	IF icschange=0 THEN
		AGBControl.eCoordSystem:=L_MC4P_CoordSystem.MCS;//笛卡尔坐标系MCS
		iCurrentCS:=L_MC4P_CoordSystem.MCS;
	END_IF
	IF icschange=1 THEN
		AGBControl.eCoordSystem:=L_MC4P_CoordSystem.ACS;//轴坐标系ACS
		iCurrentCS:=L_MC4P_CoordSystem.MCS;
	END_IF
	IF icschange=2 THEN
		AGBControl.eCoordSystem:=L_MC4P_CoordSystem.PCS_5;//PCS_5
		iCurrentCS:=L_MC4P_CoordSystem.PCS_5;
	END_IF
	IF icschange=4 THEN
		AGBControl.eCoordSystem:=L_MC4P_CoordSystem.PCS_6;//PCS_6
		iCurrentCS:=L_MC4P_CoordSystem.PCS_6;
	END_IF				
	
	AGBControl.axJogPos:=axJogPos;
	AGBControl.axJogNeg:=axJogNeg;
	xBTtest:=BYTE_TO_BOOL(bBTMenu1);
	
	//4. 读取机器人实际位置		
	ReadActPos_ACS.CoordSystem:=L_MC4P_CoordSystem.ACS;
	ReadActPos_ACS.Enable:=TRUE;
	ReadActPos_ACS(AxesGroup:=Delta_Robot);
	
	IF ReadActPos_ACS.Valid=TRUE THEN
		RobotPos.rRobotPosA1:=LREAL_TO_REAL(ReadActPos_ACS.Position[1]);
		RobotPos.rRobotPosA2:=LREAL_TO_REAL(ReadActPos_ACS.Position[2]);
		RobotPos.rRobotPosA3:=LREAL_TO_REAL(ReadActPos_ACS.Position[3]);
	END_IF

	ReadActPos_CS.CoordSystem:=iCurrentCS;
	ReadActPos_CS.Enable:=TRUE;
	ReadActPos_CS(AxesGroup:=Delta_Robot);
	
	IF ReadActPos_CS.Valid=TRUE THEN
		RobotPos.rRobotPosX:=LREAL_TO_REAL(ReadActPos_CS.Position[1]);
		RobotPos.rRobotPosY:=LREAL_TO_REAL(ReadActPos_CS.Position[2]);
		RobotPos.rRobotPosZ:=LREAL_TO_REAL(ReadActPos_CS.Position[3]);
		//RobotPos.rRobotPosC:=LREAL_TO_REAL(ReadActPos_CS.Position[7]);
		//RobotPos.rRobotPosC:=LREAL_TO_REAL(AxisYaw.lrActPosition); //modified in 2016.11.03
	END_IF
		
	//5. 机器人示教
	FOR i:=1 TO iTeachPtNO BY 1 DO				//获取当前位置
		IF bCurrentPos[i]=1 THEN
			aLRPP_TeachPoints[i].X:=RobotPos.rRobotPosX;
			aLRPP_TeachPoints[i].Y:=RobotPos.rRobotPosY;
			aLRPP_TeachPoints[i].Z:=RobotPos.rRobotPosZ;
			aLRPP_TeachPoints[i].C:=RobotPos.rRobotPosC;
			aLRPP_TeachPoints[i].CS_Num:=iCurrentCS;
			bCurrentPos[i]:=0;
		END_IF
	END_FOR
	IF bSavePt=1 THEN
			aLRPP_TeachPoints[iSelectTeNO-4].X:=RobotPos.rRobotPosX;
			aLRPP_TeachPoints[iSelectTeNO-4].Y:=RobotPos.rRobotPosY;
			aLRPP_TeachPoints[iSelectTeNO-4].Z:=RobotPos.rRobotPosZ;
			aLRPP_TeachPoints[iSelectTeNO-4].C:=RobotPos.rRobotPosC;
			aLRPP_TeachPoints[iSelectTeNO-4].CS_Num:=iCurrentCS;
			bSavePt:=0;
	END_IF
	//////////装箱示教////////
	IF xBox_ReadBelt THEN
		rBox_BeltPos:=LREAL_TO_REAL(Outfeeder.lrActPosition);
		xBox_ReadBelt:=FALSE;
	END_IF
	
	IF xBox_Tch THEN
		IF Outfeeder.lrActPosition>rBox_BeltPos THEN
			aLRPP_TeachPoints[iBox_TchNo-4].X:=LREAL_TO_REAL(RobotPos.rRobotPosX-(Outfeeder.lrActPosition-rBox_BeltPos));
		ELSE
			aLRPP_TeachPoints[iBox_TchNo-4].X:=LREAL_TO_REAL(RobotPos.rRobotPosX-(Outfeeder.lrActPosition+Outfeeder.lrcyclelength-rBox_BeltPos));
		END_IF		
		aLRPP_TeachPoints[iBox_TchNo-4].Y:=RobotPos.rRobotPosY;
		aLRPP_TeachPoints[iBox_TchNo-4].Z:=RobotPos.rRobotPosZ;
		aLRPP_TeachPoints[iBox_TchNo-4].C:=RobotPos.rRobotPosC;
		aLRPP_TeachPoints[iBox_TchNo-4].CS_Num:=iCurrentCS;
		xBox_Tch:=0;
	END_IF	

	//装箱体初始化
	p_rBoxLength:=rBoxLength;				//箱体长度
	p_rBoxBiasLength:=rBoxBiasLength;		//箱体偏置长度//产品检测传感器初始化

	p_iNewProdNum:=iNewProdNum;
	//检测产品传感器设置
 
	p_rBoxOutfeederVel:=rBoxOutfeederVel;// 装箱时出料带的速度
	p_rBoxPickTime:=rBoxPickTime;// 装箱抓取物料时间
	p_rBoxPlaceTime:=rBoxPlaceTime;// 装箱放置物料时间
	p_rBoxDetectPosX:=rBoxDetectPosX;// 装箱检测箱体的初始位置     
	p_iBoxTotalPrdoNr:=iBoxTotalPrdoNr;
	//////////装箱示教////////
	
	
	//6. 吸盘标定		

	IF xReadCalibCaxisAngle THEN
		rCalibCaxisAngle:=LREAL_TO_REAL(RobotPos.rRobotPosC);
		rCalibCaxisAngletoRad:=LREAL_TO_REAL(rCalibCaxisAngle*2*Pi/360);
	END_IF

												
	p_iSuckerNum:=iSuckerNum; 	//吸盘标定
	p_iCalibSucker:=iCalibSucker;
	p_rSuker1BiasX:=rSuker1BiasX;
	p_rSuker1BiasY:=rSuker1BiasY;
	p_rSuker2BiasX:=rSuker2BiasX;
	p_rSuker2BiasY:=rSuker2BiasY;
	p_rSuker3BiasX:=rSuker3BiasX;
	p_rSuker3BiasY:=rSuker3BiasY;
	p_rSuker4BiasX:=rSuker4BiasX;
	p_rSuker4BiasY:=rSuker4BiasY;
	//p_rCalibCaxisAngle:=rCalibCaxisAngle;	
		
	IF xToolActive THEN	
		xToolActive:=FALSE;		
	END_IF	
	
	IF 	xToolDeActive THEN
		xToolDeActive:=FALSE;
	END_IF
		
	IF iCalibSucker=0 THEN
		rBiasX:=0;
		rBiasY:=0;	
	END_IF
	IF iCalibSucker=1 THEN
		rBiasX:=rSuker1BiasX;
		rBiasY:=rSuker1BiasY;	
	END_IF
	
	IF iCalibSucker=2 THEN
		rBiasX:=rSuker2BiasX;
		rBiasY:=rSuker2BiasY;	
	END_IF	

	IF iCalibSucker=3 THEN
		rBiasX:=rSuker3BiasX;
		rBiasY:=rSuker3BiasY;				
	END_IF		
	
	IF iCalibSucker=4 THEN
		rBiasX:=rSuker4BiasX;
		rBiasY:=rSuker4BiasY;				
	END_IF	
         
	
	//7. InfeedBeltOrigin坐标系标定
	IF xInfeedRead0=TRUE THEN
		p_rConveyorInRecord0:=rConveyorInRecord0:=LREAL_TO_REAL(Infeeder.lrActPosition);
	END_IF
	p_rConveyorInRecord0:=rConveyorInRecord0;
	
	IF xInfeedRead1=TRUE THEN
		IF Infeeder.lrActPosition<rConveyorInRecord0 THEN
			p_rConveyorInRecord1:=rConveyorInRecord1:=LREAL_TO_REAL(Infeeder.lrActPosition+Infeeder.lrcyclelength);
		ELSE
			p_rConveyorInRecord1:=rConveyorInRecord1:=LREAL_TO_REAL(Infeeder.lrActPosition);
		END_IF		
		p_rReadInfeedPos1_X:=rReadInfeedPos1_X:=LREAL_TO_REAL(RobotPos.rRobotPosX);
		p_rReadInfeedPos1_Y:=rReadInfeedPos1_Y:=LREAL_TO_REAL(RobotPos.rRobotPosY);
		p_rReadInfeedPos1_Z:=rReadInfeedPos1_Z:=LREAL_TO_REAL(RobotPos.rRobotPosZ);
	END_IF
	p_rConveyorInRecord1:=rConveyorInRecord1;
	p_rReadInfeedPos1_X:=rReadInfeedPos1_X;
	p_rReadInfeedPos1_Y:=rReadInfeedPos1_Y;
	p_rReadInfeedPos1_Z:=rReadInfeedPos1_Z;
	
	IF xInfeedRead2=TRUE THEN
		IF Infeeder.lrActPosition<rConveyorInRecord1 THEN
			p_rConveyorInRecord2:=rConveyorInRecord2:=LREAL_TO_REAL(Infeeder.lrActPosition+Infeeder.lrcyclelength);
		ELSE
			p_rConveyorInRecord2:=rConveyorInRecord2:=LREAL_TO_REAL(Infeeder.lrActPosition);
		END_IF

		p_rReadInfeedPos2_X:=rReadInfeedPos2_X:=LREAL_TO_REAL(RobotPos.rRobotPosX);
		p_rReadInfeedPos2_Y:=rReadInfeedPos2_Y:=LREAL_TO_REAL(RobotPos.rRobotPosY);
		p_rReadInfeedPos2_Z:=rReadInfeedPos2_Z:=LREAL_TO_REAL(rReadInfeedPos1_Z);//标定与Z无关，仅取一次Z值		
	END_IF
	
	p_rConveyorInRecord2:=rConveyorInRecord2;
	p_rReadInfeedPos2_X:=rReadInfeedPos2_X;
	p_rReadInfeedPos2_Y:=rReadInfeedPos2_Y;
	p_rReadInfeedPos2_Z:=rReadInfeedPos2_Z;
	
	IF xInfeedRead3=TRUE THEN
		p_rReadInfeedPos3_X:=rReadInfeedPos3_X:=LREAL_TO_REAL(RobotPos.rRobotPosX);
		p_rReadInfeedPos3_Y:=rReadInfeedPos3_Y:=LREAL_TO_REAL(RobotPos.rRobotPosY);
		p_rReadInfeedPos3_Z:=rReadInfeedPos3_Z:=LREAL_TO_REAL(rReadInfeedPos1_Z);//标定与Z无关，仅取一次Z值		
	END_IF
	
	
	p_rReadInfeedPos3_X:=rReadInfeedPos3_X;
	p_rReadInfeedPos3_Y:=rReadInfeedPos3_Y;
	p_rReadInfeedPos3_Z:=rReadInfeedPos3_Z;
	
	IF xInfeedRead4=TRUE THEN
		p_rReadInfeedPos4_X:=rReadInfeedPos4_X:=LREAL_TO_REAL(RobotPos.rRobotPosX);
		p_rReadInfeedPos4_Y:=rReadInfeedPos4_Y:=LREAL_TO_REAL(RobotPos.rRobotPosY);
		p_rReadInfeedPos4_Z:=rReadInfeedPos4_Z:=LREAL_TO_REAL(rReadInfeedPos1_Z);//标定与Z无关，仅取一次Z值		
	END_IF
	
	p_rReadInfeedPos4_X:=rReadInfeedPos4_X;
	p_rReadInfeedPos4_Y:=rReadInfeedPos4_Y;
	p_rReadInfeedPos4_Z:=rReadInfeedPos4_Z;		

	//计算传动带（进料带）原点并标定PCS5（InS）
	IF xCaculateInfeedBeltOrigin=TRUE THEN
		
		FourPts_Calibration_1(
			rReadfeedPos1_X:= rReadInfeedPos1_X, 
			rReadfeedPos1_Y:= rReadInfeedPos1_Y, 
			rReadfeedPos1_Z:= rReadInfeedPos1_Z, 
			rReadfeedPos2_X:= rReadInfeedPos2_X, 
			rReadfeedPos2_Y:= rReadInfeedPos2_Y, 
			rReadfeedPos3_X:= rReadInfeedPos3_X, 
			rReadfeedPos3_Y:= rReadInfeedPos3_Y, 
			rReadfeedPos4_X:= rReadInfeedPos4_X, 
			rReadfeedPos4_Y:= rReadInfeedPos4_Y, 
			rRotation_C=> sInFeedBeltOrigin.rRotation_C,
			Output_X0=>PCS5_X0	,
			Output_Y0=>PCS5_Y0	,	
			Output_X1=>PCS5_X1	,	
			Output_Y1=>PCS5_Y1	,	
			Output_X2=>PCS5_X2	,	
			Output_Y2=>PCS5_Y2	,	
			Output_X3=>PCS5_X3	,	
			Output_Y3=>PCS5_Y3	,	
			dx=>PCS5_dx	,			
			dy=>PCS5_dy	,	);
			  	
		p_PCS5_X0:=PCS5_X0;
		p_PCS5_Y0:=PCS5_Y0;
		p_PCS5_X1:=PCS5_X1;
		p_PCS5_Y1:=PCS5_Y1;
		p_PCS5_X2:=PCS5_X2;
		p_PCS5_Y2:=PCS5_Y2;
		p_PCS5_X3:=PCS5_X3;
		p_PCS5_Y3:=PCS5_Y3;
		p_PCS5_dx:=PCS5_dx;
		p_PCS5_dy:=PCS5_dy;
		
		//p_sInFeedBeltOrigin.rOriginPosX:=sInFeedBeltOrigin.rOriginPosX:=rReadInfeedPos1_X;
		//p_sInFeedBeltOrigin.rOriginPosY:=sInFeedBeltOrigin.rOriginPosY:=rReadInfeedPos1_Y;
		p_sInFeedBeltOrigin.rOriginPosX:=sInFeedBeltOrigin.rOriginPosX:=(rReadInfeedPos1_X+rReadInfeedPos2_X+rReadInfeedPos3_X+rReadInfeedPos4_X)/4.0;
		p_sInFeedBeltOrigin.rOriginPosY:=sInFeedBeltOrigin.rOriginPosY:=(rReadInfeedPos1_Y+rReadInfeedPos2_Y+rReadInfeedPos3_Y+rReadInfeedPos4_Y)/4.0;
		
		p_sInFeedBeltOrigin.rOriginPosZ:=sInFeedBeltOrigin.rOriginPosZ:=rReadInfeedPos1_Z;
		p_sInFeedBeltOrigin.rRotation_C:=sInFeedBeltOrigin.rRotation_C;
						
		//开始标定InS（PCS5）			
		fbPCS5_Calib.TransX:=p_PCS5_OriginX:=PCS5_OriginX:=	p_sInFeedBeltOrigin.rOriginPosX;
		fbPCS5_Calib.TransY:=p_PCS5_OriginY:=PCS5_OriginY:=	p_sInFeedBeltOrigin.rOriginPosY;
		fbPCS5_Calib.TransZ:=p_PCS5_OriginZ:=PCS5_OriginZ:=	p_sInFeedBeltOrigin.rOriginPosZ;
		fbPCS5_Calib.RotAngle1:=p_PCS5_OriginA:=PCS5_OriginA:=	p_sInFeedBeltOrigin.rRotation_A;
		fbPCS5_Calib.RotAngle2:=p_PCS5_OriginB:=PCS5_OriginB:=	p_sInFeedBeltOrigin.rRotation_B;
		fbPCS5_Calib.RotAngle3:=p_PCS5_OriginC:=PCS5_OriginC:=	p_sInFeedBeltOrigin.rRotation_C;
		fbPCS5_Calib.Execute:=TRUE;
		fbPCS5_Calib.CoordSystem:=L_MC4P_CoordSystem.PCS_5;	
		xCaculateInfeedBeltOrigin:=FALSE;
		
	END_IF
	
	IF fbPCS5_Calib.Done=TRUE THEN
		fbPCS5_Calib.Execute:=FALSE;
	END_IF			
	fbPCS5_Calib(AxesGroup:=Delta_Robot);

	
	//再次将标定值赋给Pst，以便用户自修改	
	p_sInFeedBeltOrigin.rOriginPosX:=sInFeedBeltOrigin.rOriginPosX; //传动带原点
	p_sInFeedBeltOrigin.rOriginPosY:=sInFeedBeltOrigin.rOriginPosY;
	p_sInFeedBeltOrigin.rOriginPosZ:=sInFeedBeltOrigin.rOriginPosZ;
	p_sInFeedBeltOrigin.rRotation_A:=sInFeedBeltOrigin.rRotation_A;
	p_sInFeedBeltOrigin.rRotation_B:=sInFeedBeltOrigin.rRotation_B;
	p_sInFeedBeltOrigin.rRotation_C:=sInFeedBeltOrigin.rRotation_C;
	
			
	//8. OutfeedBeltOrigin坐标系标定 Outfeeder是出料带
	IF xOutfeedRead0=TRUE THEN
		p_rConveyorOutRecord0:=rConveyorOutRecord0:=LREAL_TO_REAL(Outfeeder.lrActPosition);
	END_IF
	
	p_rConveyorOutRecord0:=rConveyorOutRecord0;
	
	IF xOutfeedRead1=TRUE THEN
		IF Outfeeder.lrActPosition<rConveyorOutRecord0 THEN
			p_rConveyorOutRecord1:=rConveyorOutRecord1:=LREAL_TO_REAL(Outfeeder.lrActPosition+Outfeeder.lrcyclelength);
		ELSE
			p_rConveyorOutRecord1:=rConveyorOutRecord1:=LREAL_TO_REAL(Outfeeder.lrActPosition);
		END_IF	
		p_rReadOutfeedPos1_X:=rReadOutfeedPos1_X:=LREAL_TO_REAL(RobotPos.rRobotPosX);
		p_rReadOutfeedPos1_Y:=rReadOutfeedPos1_Y:=LREAL_TO_REAL(RobotPos.rRobotPosY);
		p_rReadOutfeedPos1_Z:=rReadOutfeedPos1_Z:=LREAL_TO_REAL(RobotPos.rRobotPosZ);
	END_IF
	p_rConveyorOutRecord1:=rConveyorOutRecord1;
	p_rReadOutfeedPos1_X:=rReadOutfeedPos1_X;
	p_rReadOutfeedPos1_Y:=rReadOutfeedPos1_Y;
	p_rReadOutfeedPos1_Z:=rReadOutfeedPos1_Z;		
	                            
	IF xOutfeedRead2=TRUE THEN
		IF Outfeeder.lrActPosition<rConveyorOutRecord1 THEN
			p_rConveyorOutRecord2:=rConveyorOutRecord2:=LREAL_TO_REAL(Outfeeder.lrActPosition+Outfeeder.lrcyclelength);
		ELSE
			p_rConveyorOutRecord2:=rConveyorOutRecord2:=LREAL_TO_REAL(Outfeeder.lrActPosition);
		END_IF	

		p_rReadOutfeedPos2_X:=rReadOutfeedPos2_X:=LREAL_TO_REAL(RobotPos.rRobotPosX);
		p_rReadOutfeedPos2_Y:=rReadOutfeedPos2_Y:=LREAL_TO_REAL(RobotPos.rRobotPosY);
		p_rReadOutfeedPos2_Z:=rReadOutfeedPos2_Z:=LREAL_TO_REAL(rReadOutfeedPos1_Z);//标定与Z无关，仅取一次Z值
	END_IF
	p_rConveyorOutRecord2:=rConveyorOutRecord2;
	p_rReadOutfeedPos2_X:=rReadOutfeedPos2_X;
	p_rReadOutfeedPos2_Y:=rReadOutfeedPos2_Y;	
	p_rReadOutfeedPos2_Z:=rReadOutfeedPos2_Z;	
	
	IF xOutfeedRead3=TRUE THEN
		p_rReadOutfeedPos3_X:=rReadOutfeedPos3_X:=LREAL_TO_REAL(RobotPos.rRobotPosX);
		p_rReadOutfeedPos3_Y:=rReadOutfeedPos3_Y:=LREAL_TO_REAL(RobotPos.rRobotPosY);
		p_rReadOutfeedPos3_Z:=rReadOutfeedPos3_Z:=LREAL_TO_REAL(rReadOutfeedPos1_Z);//标定与Z无关，仅取一次Z值
	END_IF

	p_rReadOutfeedPos3_X:=rReadOutfeedPos3_X;
	p_rReadOutfeedPos3_Y:=rReadOutfeedPos3_Y;	
	p_rReadOutfeedPos3_Z:=rReadOutfeedPos3_Z;	
	
	IF xOutfeedRead4=TRUE THEN
		p_rReadOutfeedPos4_X:=rReadOutfeedPos4_X:=LREAL_TO_REAL(RobotPos.rRobotPosX);
		p_rReadOutfeedPos4_Y:=rReadOutfeedPos4_Y:=LREAL_TO_REAL(RobotPos.rRobotPosY);
		p_rReadOutfeedPos4_Z:=rReadOutfeedPos4_Z:=LREAL_TO_REAL(rReadOutfeedPos1_Z);//标定与Z无关，仅取一次Z值
	END_IF
	
	p_rReadOutfeedPos4_X:=rReadOutfeedPos4_X;
	p_rReadOutfeedPos4_Y:=rReadOutfeedPos4_Y;	
	p_rReadOutfeedPos4_Z:=rReadOutfeedPos4_Z;	

	
	//计算传动带（出料带）原点并标定PCS6（OtS）
	IF	xCaculateOutfeedBeltOrigin=TRUE THEN
		
			FourPts_Calibration_2(
					rReadfeedPos1_X:= rReadOutfeedPos1_X, 
					rReadfeedPos1_Y:= rReadOutfeedPos1_Y, 
					rReadfeedPos1_Z:= rReadOutfeedPos1_Z, 
					rReadfeedPos2_X:= rReadOutfeedPos2_X, 
					rReadfeedPos2_Y:= rReadOutfeedPos2_Y, 
					rReadfeedPos3_X:= rReadOutfeedPos3_X, 
					rReadfeedPos3_Y:= rReadOutfeedPos3_Y, 
					rReadfeedPos4_X:= rReadOutfeedPos4_X, 
					rReadfeedPos4_Y:= rReadOutfeedPos4_Y, 
					rRotation_C=> sOutFeedBeltOrigin.rRotation_C,
					Output_X0=>PCS6_X0	,
                    Output_Y0=>PCS6_Y0	,	
                    Output_X1=>PCS6_X1	,	
                    Output_Y1=>PCS6_Y1	,	
                    Output_X2=>PCS6_X2	,	
                    Output_Y2=>PCS6_Y2	,	
                    Output_X3=>PCS6_X3	,	
                    Output_Y3=>PCS6_Y3	,	
               		dx=>PCS6_dx	,			
			        dy=>PCS6_dy	,	);
			  	
			p_PCS6_X0:=PCS6_X0;
			p_PCS6_Y0:=PCS6_Y0;
			p_PCS6_X1:=PCS6_X1;
			p_PCS6_Y1:=PCS6_Y1;
			p_PCS6_X2:=PCS6_X2;
			p_PCS6_Y2:=PCS6_Y2;
			p_PCS6_X3:=PCS6_X3;
			p_PCS6_Y3:=PCS6_Y3;
			p_PCS6_dx:=PCS6_dx;
			p_PCS6_dy:=PCS6_dy;
			
			p_sOutFeedBeltOrigin.rOriginPosX:=sOutFeedBeltOrigin.rOriginPosX:=(rReadOutfeedPos1_X+rReadOutfeedPos2_X+rReadOutfeedPos3_X+rReadOutfeedPos4_X)/4.0;
			p_sOutFeedBeltOrigin.rOriginPosY:=sOutFeedBeltOrigin.rOriginPosY:=(rReadOutfeedPos1_Y+rReadOutfeedPos2_Y+rReadOutfeedPos3_Y+rReadOutfeedPos4_Y)/4.0;
			//p_sOutFeedBeltOrigin.rOriginPosX:=sOutFeedBeltOrigin.rOriginPosX:=rReadOutfeedPos1_X;
			//p_sOutFeedBeltOrigin.rOriginPosY:=sOutFeedBeltOrigin.rOriginPosY:=rReadOutfeedPos1_Y;
			p_sOutFeedBeltOrigin.rOriginPosZ:=sOutFeedBeltOrigin.rOriginPosZ:=rReadOutfeedPos1_Z;
			p_sOutFeedBeltOrigin.rRotation_C:=sOutFeedBeltOrigin.rRotation_C;
			
			//开始标定InS（PCS5）
			fbPCS6_Calib.TransX:=p_PCS6_OriginX:=PCS6_OriginX:=p_sOutFeedBeltOrigin.rOriginPosX;
			fbPCS6_Calib.TransY:=p_PCS6_OriginY:=PCS6_OriginY:=p_sOutFeedBeltOrigin.rOriginPosY;
			fbPCS6_Calib.TransZ:=p_PCS6_OriginZ:=PCS6_OriginZ:=p_sOutFeedBeltOrigin.rOriginPosZ;
			fbPCS6_Calib.RotAngle1:=p_PCS6_OriginA:=PCS6_OriginA:=p_sOutFeedBeltOrigin.rRotation_A;
			fbPCS6_Calib.RotAngle2:=p_PCS6_OriginB:=PCS6_OriginB:=p_sOutFeedBeltOrigin.rRotation_B;
			fbPCS6_Calib.RotAngle3:=p_PCS6_OriginC:=PCS6_OriginC:=p_sOutFeedBeltOrigin.rRotation_C;
			fbPCS6_Calib.Execute:=TRUE;
			fbPCS6_Calib.CoordSystem:=L_MC4P_CoordSystem.PCS_6;	
			xCaculateOutfeedBeltOrigin:=FALSE;
			
	END_IF
	
	IF fbPCS6_Calib.Done=TRUE THEN
		fbPCS6_Calib.Execute:=FALSE;
	END_IF
	fbPCS6_Calib(AxesGroup:=Delta_Robot);	
	//出料带标定模块
	
	
	
	//再次将标定值赋给Pst，以便用户自修改	
	p_sOutFeedBeltOrigin.rOriginPosX:=sOutFeedBeltOrigin.rOriginPosX; //传动带原点
	p_sOutFeedBeltOrigin.rOriginPosY:=sOutFeedBeltOrigin.rOriginPosY;
	p_sOutFeedBeltOrigin.rOriginPosZ:=sOutFeedBeltOrigin.rOriginPosZ;
	p_sOutFeedBeltOrigin.rRotation_A:=sOutFeedBeltOrigin.rRotation_A;
	p_sOutFeedBeltOrigin.rRotation_B:=sOutFeedBeltOrigin.rRotation_B;
	p_sOutFeedBeltOrigin.rRotation_C:=sOutFeedBeltOrigin.rRotation_C;

	//9. 相机标定界面
	IF xTeachRCalPt2 THEN
		p_RobotCalPt2.rX:=RobotCalPt2.rX:=RobotPos.rRobotPosX+rInfeedMapX;
		p_RobotCalPt2.rY:=RobotCalPt2.rY:=RobotPos.rRobotPosY+rInfeedMapY;
		p_RobotCalPt2.rZ:=RobotCalPt2.rZ:=RobotPos.rRobotPosZ;		
	END_IF
	
	IF xTeachRCalPt3 THEN
		p_RobotCalPt3.rX:=RobotCalPt3.rX:=RobotPos.rRobotPosX+rInfeedMapX;
		p_RobotCalPt3.rY:=RobotCalPt3.rY:=RobotPos.rRobotPosY+rInfeedMapY;
		p_RobotCalPt3.rZ:=RobotCalPt3.rZ:=RobotPos.rRobotPosZ;		
	END_IF																	
	IF xTeachRCalPt4 THEN
		p_RobotCalPt4.rX:=RobotCalPt4.rX:=RobotPos.rRobotPosX+rInfeedMapX;
		p_RobotCalPt4.rY:=RobotCalPt4.rY:=RobotPos.rRobotPosY+rInfeedMapY;
		p_RobotCalPt4.rZ:=RobotCalPt4.rZ:=RobotPos.rRobotPosZ;		
	END_IF	
	
	IF xCaculateCameraCalPts THEN
		
		p_CameraCalPt1.rX:=CameraCalPt1.rX:=(RobotCalPt1.rX-sInFeedBeltOrigin.rOriginPosX)*COS(alpha)+(RobotCalPt1.rY-sInFeedBeltOrigin.rOriginPosY)*SIN(alpha)-(rConveyorInRecord2-rConveyorInRecord0);
		p_CameraCalPt1.rY:=CameraCalPt1.rY:=(-RobotCalPt1.rX+sInFeedBeltOrigin.rOriginPosX)*SIN(alpha)+(RobotCalPt1.rY-sInFeedBeltOrigin.rOriginPosY)*COS(alpha);//-(rConveyorInRecord2-rConveyorInRecord0);
		p_CameraCalPt1.rZ:=CameraCalPt1.rZ:=0;
		
		p_CameraCalPt2.rX:=CameraCalPt2.rX:=(RobotCalPt2.rX-sInFeedBeltOrigin.rOriginPosX)*COS(alpha)+(RobotCalPt2.rY-sInFeedBeltOrigin.rOriginPosY)*SIN(alpha)-(rConveyorInRecord2-rConveyorInRecord0);
		p_CameraCalPt2.rY:=CameraCalPt2.rY:=(-RobotCalPt2.rX+sInFeedBeltOrigin.rOriginPosX)*SIN(alpha)+(RobotCalPt2.rY-sInFeedBeltOrigin.rOriginPosY)*COS(alpha);//-(rConveyorInRecord2-rConveyorInRecord0);
		p_CameraCalPt2.rZ:=CameraCalPt2.rZ:=0;
		
		p_CameraCalPt3.rX:=CameraCalPt3.rX:=(RobotCalPt3.rX-sInFeedBeltOrigin.rOriginPosX)*COS(alpha)+(RobotCalPt3.rY-sInFeedBeltOrigin.rOriginPosY)*SIN(alpha)-(rConveyorInRecord2-rConveyorInRecord0);
		p_CameraCalPt3.rY:=CameraCalPt3.rY:=(-RobotCalPt3.rX+sInFeedBeltOrigin.rOriginPosX)*SIN(alpha)+(RobotCalPt3.rY-sInFeedBeltOrigin.rOriginPosY)*COS(alpha);//-(rConveyorInRecord2-rConveyorInRecord0);
		p_CameraCalPt3.rZ:=CameraCalPt3.rZ:=0;
		
		p_CameraCalPt4.rX:=CameraCalPt4.rX:=(RobotCalPt4.rX-sInFeedBeltOrigin.rOriginPosX)*COS(alpha)+(RobotCalPt4.rY-sInFeedBeltOrigin.rOriginPosY)*SIN(alpha)-(rConveyorInRecord2-rConveyorInRecord0);
		p_CameraCalPt4.rY:=CameraCalPt4.rY:=(-RobotCalPt4.rX+sInFeedBeltOrigin.rOriginPosX)*SIN(alpha)+(RobotCalPt4.rY-sInFeedBeltOrigin.rOriginPosY)*COS(alpha);//-(rConveyorInRecord2-rConveyorInRecord0);
		p_CameraCalPt4.rZ:=CameraCalPt4.rZ:=0;
	
	END_IF
		
END_IF		

(*

IF xAutoRun  or xJumpOutManualJog THEN
	wstep:=5;//返回待机状态
	xJumpOutManualJog:=FALSE;
END_IF

*)
END_ACTION

ACTION A30_AutoRun:
	CustomerPrgHandling.xEnable:=xAutoRun;
IF xAutoRun THEN
	IF iSelfadaptPickSwitch=1 THEN
		lrMaxTimeforCycleAdaptive:=1.0;
	ELSE
		lrMaxTimeforCycleAdaptive:=0.0;
	END_IF
	// 抓取节拍自适应计算
	
	//传送带滤波处理
	L_USPP_PT1Filter_0(
		lrIn:= , 
		lrDelayTime:=1.0 , 
		lrOut=> lrInfeederFilterVelocity, 
		xError=> , 
		eErrorID=> );		
	lrDistToMinCapLForCycleAdaptive:=lrInfeederFilterVelocity*lrMaxTimeforCycleAdaptive;		
	//传送带滤波处理
	
	p_xExternalMode:=xExternalMode;//将外部数据发送模式赋值到断电保持变量 3.1
	
	p_xLocal_or_Remote:=xLocal_or_Remote; //机器人本机控制 or 远程控制
	
	IF fb_PlaceCounter_Triger.Q THEN
		iPlaceCounter:=iPlaceCounter+1;
	END_IF
	
	//托盘的x、y方向间距设置===================2017.12.13============================
		CustomerPrgHandling.rPalletPickDeltaX:=PCS5_dx;
		CustomerPrgHandling.rPalletPickDeltaY:=PCS5_dy;
		CustomerPrgHandling.rPalletPlaceDeltaX:=PCS6_dx;
		CustomerPrgHandling.rPalletPlaceDeltaY:=PCS6_dy;
	//托盘的x、y方向间距设置===================2017.12.13============================	
		
	//抓取线和放置线的计算
	rMinCaptureLine:=CustomerPrg.Table_Position[5].X;
	rMaxCaptureLine:=CustomerPrg.Table_Position[6].X;
	rMinPlaceLine:=CustomerPrg.Table_Position[7].X;
	rMaxPlaceLine:=CustomerPrg.Table_Position[8].X;
	//产品信息
	rProductAdd_Z:=CustomerPrg.Table_Position[9].Z;			
	rFilterTolerance_X:=CustomerPrg.Table_Position[9].X;
	rFilterTolerance_Y:=CustomerPrg.Table_Position[9].Y;	
	
	
	//程序解析运动函数
	//程序解析模块输入	
	//2017.03.30  PnP Cycle Adaptive Fuction
	CustomerPrgHandling.lrDistToMinCapLForCycleAdaptive:=lrDistToMinCapLForCycleAdaptive;
	CustomerPrgHandling.lrMinCaptureLine:= rMinCaptureLine;
	CustomerPrgHandling.lrMaxCaptureLine:= rMaxCaptureLine; 
	
	(*
	CustomerPrgHandling.rCoefMaxOfStartAndEndR[1]:=CoefMaxOfStartAndEndR[1];
	CustomerPrgHandling.iAux1ExePointPassed[1]:=Aux1ExePointPassed[1];		
	CustomerPrgHandling.rAux1DurationRatio[1]:=Aux1DurationRatio[1];				
	CustomerPrgHandling.iAux1MotionLaw[1]:=Aux1MotionLaw[1];				
	CustomerPrgHandling.rStartAlphaRatio[1,1]:=StartAlphaRatio[1,1];	
	CustomerPrgHandling.rStartAlphaRatio[1,2]:=StartAlphaRatio[1,2];
	CustomerPrgHandling.rStartAlphaRatio[1,3]:=StartAlphaRatio[1,3];		
	CustomerPrgHandling.rEndAlphaRatio[1,7]:=EndAlphaRatio[1,7];
	CustomerPrgHandling.rEndAlphaRatio[1,8]:=EndAlphaRatio[1,8];
	CustomerPrgHandling.rEndAlphaRatio[1,9]:=EndAlphaRatio[1,9];
	
	CustomerPrgHandling.rCoefMaxOfStartAndEndR[2]:= CoefMaxOfStartAndEndR[2];
	CustomerPrgHandling.iAux1ExePointPassed[2]:= Aux1ExePointPassed[2];		
	CustomerPrgHandling.rAux1DurationRatio[2]:= Aux1DurationRatio[2];				
	CustomerPrgHandling.iAux1MotionLaw[2]:=Aux1MotionLaw[2];				
	CustomerPrgHandling.rStartAlphaRatio[2,1]:=StartAlphaRatio[2,1];	
	CustomerPrgHandling.rStartAlphaRatio[2,2]:=StartAlphaRatio[2,2];
	CustomerPrgHandling.rStartAlphaRatio[2,3]:=StartAlphaRatio[2,3];		
	CustomerPrgHandling.rEndAlphaRatio[2,7]:=EndAlphaRatio[2,7];
	CustomerPrgHandling.rEndAlphaRatio[2,8]:=EndAlphaRatio[2,8];
	CustomerPrgHandling.rEndAlphaRatio[2,9]:=EndAlphaRatio[2,9];
	*)
		
	CustomerPrgHandling.xDetectBoxSwitch:=DI_3;
	CustomerPrgHandling.CustomerPrg:=CustomerPrg;
	CustomerPrgHandling.xRunInter:=xRunInter;
	CustomerPrgHandling.xStopInter:=xStopInter;
	CustomerPrgHandling.sInFeedBeltOrigin:=	sInFeedBeltOrigin;	
	CustomerPrgHandling.sOutFeedBeltOrigin:=sOutFeedBeltOrigin;                                                            
	//CustomerPrgHandling.lrCurrentAuxC:=AxisYaw.lrActPosition;
	CustomerPrgHandling.rFollowBias_X:=rFollowBias_X;//1
	CustomerPrgHandling.rFollowBias_Y:=rFollowBias_Y;//2
	CustomerPrgHandling.rSuckerDropHeight:=rSuckerDropHeight;//3
	CustomerPrgHandling.rInfeedClutchPra:=rBelt1_ClutchPra;//4
	CustomerPrgHandling.rOutfeedClutchPra:=rBelt2_ClutchPra;//5
	CustomerPrgHandling.rBlowOpenTime:=	rBlow_Gas_OpenTime;//6
	CustomerPrgHandling.rSuckOpenTime:=rSuck_Gas_OpenTime;//7
	CustomerPrgHandling.rBlowGasTime:=rBlowGasTime;//8	
	CustomerPrgHandling.iBox_ExceptionDeal:=iBox_ExceptionDeal;//9
	CustomerPrgHandling.iSelfadaptPickSwitch:=iSelfadaptPickSwitch;//10
	CustomerPrgHandling.rPnPDurationNegativeLimit:=rPnPDurationNegativeLimit;
	CustomerPrgHandling.rPnPDurationPositiveLimit:=rPnPDurationPositiveLimit;	
	CustomerPrgHandling.iProdDeformation:=iProdDeformation; //11 产品变形量	

	CustomerPrgHandling.rProductAdd_Z:=rProductAdd_Z;
	CustomerPrgHandling.rBoxLength:=rBoxLength;
	CustomerPrgHandling.rBoxBiasLength:=rBoxBiasLength;
	
	CustomerPrgHandling.iNewProdNum:=iNewProdNum;//检测物体需要的外部触发信号数量
	
	IF iPrdtDetectDevice=Detect_Device.Camera THEN//产品检测装置选择 	0：相机；1：传感器；2：上位机通讯指定	 可以定义成枚举类型
		IF iSuckerNum <=5 THEN
			CustomerPrgHandling.xProdInfoReady:=BufferHandling.xProdInfoReady;
			CustomerPrgHandling.lrInfeedDeltaX:=BufferHandling.sFirstProdInfo.lrDeltaX;
			CustomerPrgHandling.lrInfeedDeltaY:=BufferHandling.sFirstProdInfo.lrDeltaY;
			CustomerPrgHandling.lrPosAuxC:=BufferHandling.sFirstProdInfo.lrPosAuxC;			
		ELSIF iSuckerNum >=6 THEN		
			CustomerPrgHandling.xProdInfoReady:=MultiPickHandling.xProdGroupReady AND MultiPickHandling.xProdInfoReady;			
			CustomerPrgHandling.lrInfeedDeltaX:=MultiPickHandling.sProductInfo.lrDeltaX;
			CustomerPrgHandling.lrInfeedDeltaY:=MultiPickHandling.sProductInfo.lrDeltaY;
			CustomerPrgHandling.lrPosAuxC:=MultiPickHandling.sProductInfo.lrPosAuxC;		
		END_IF	
	END_IF
	
	IF iPrdtDetectDevice=Detect_Device.Sensor THEN//产品检测装置选择 0：相机；1：传感器；2：上位机通讯指定	
		CustomerPrgHandling.xProdInfoReady:=SensorBufferHandler.xProdInfoReady;
		CustomerPrgHandling.lrInfeedDeltaX:=SensorBufferHandler.sFirstProdInfo.lrDeltaX;
		CustomerPrgHandling.lrInfeedDeltaY:=SensorBufferHandler.sFirstProdInfo.lrDeltaY;
		CustomerPrgHandling.lrPosAuxC:=SensorBufferHandler.sFirstProdInfo.lrPosAuxC;
	END_IF
	
	//程序解析模块输出
	iCommandType							:=CustomerPrgHandling.iCommandType;
	iCurrentPrgCmdNum						:=CustomerPrgHandling.iCurrentPrgCmdNum;
	LoadDistribution.lrFilterTolerance		:=rFilterTolerance_X; //滤波参数
	
	BufferHandling.xFirstProdDel			:=CustomerPrgHandling.xFirstProdDel;
	BufferHandling.lrPaPDuration			:=CustomerPrgHandling.lrPaPDuration;	
	BufferHandling.lrMinCaptureLine			:=rMinCaptureLine;	//抓取起始线	
	BufferHandling.lrMaxCaptureLine			:=rMaxCaptureLine;	//抓取起始线     	
	
	MultiPickHandling.xProductDel			:=CustomerPrgHandling.xFirstProdDel;
	MultiPickHandling.lrPaPDuration			:=CustomerPrgHandling.lrPaPDuration;
	MultiPickHandling.lrMinCaptureLine		:=rMinCaptureLine;	//抓取线限位1 
	MultiPickHandling.lrMaxCaptureLine		:=rMaxCaptureLine;	//抓取线限位2
	MultiPickHandling.lrToleranceDistance	:=500;
	MultiPickHandling.iNrOfTool				:=iSuckerNum;
	
	(*
	xProdInfoReady_TON(IN:=MultiPickHandling.xProdInfoReady,Pt:=T#50MS);
	IF xProdInfoReady_TON.Q THEN
		MultiPickHandling.xProductDel:=TRUE;	
	END_IF
	xProductDel_TON(IN:=MultiPickHandling.xProductDel,Pt:=T#4MS);
	IF xProductDel_TON.Q THEN
		MultiPickHandling.xProductDel:=FALSE;
	END_IF
	*)
	
	//吸气/吹气
	//x_Suck1:=CustomerPrgHandling.xSuck;
	//x_Blow1:=CustomerPrgHandling.xBlow;
	IF xAutoRun THEN
		x_Suck1_HMI:=FALSE;
		x_Blow1_HMI:=FALSE;
	END_IF
	
	
	//传感器检测输入
	SensorBufferHandler.lrMinPickLine:=rMinCaptureLine;
	SensorBufferHandler.lrMaxPickLine:=rMaxCaptureLine;
	SensorBufferHandler.lrPaPDuration:=CustomerPrgHandling.lrPaPDuration;
	SensorBufferHandler.xFirstProdDel:=CustomerPrgHandling.xFirstProdDel;
	
	//传入工具坐标系参数
	CustomerPrgHandling.Tool[1].X:=rSuker1BiasX;
	CustomerPrgHandling.Tool[1].Y:=rSuker1BiasY;
	CustomerPrgHandling.Tool[1].C:=rSuker1PickC;
	//CustomerPrgHandling.Tool[1].Z:=iSuckerHeight;
	CustomerPrgHandling.Tool[2].X:=rSuker2BiasX;
	CustomerPrgHandling.Tool[2].Y:=rSuker2BiasY;
	CustomerPrgHandling.Tool[2].C:=rSuker2PickC;
	//CustomerPrgHandling.Tool[2].Z:=iSuckerHeight;
	CustomerPrgHandling.Tool[3].X:=rSuker3BiasX;
	CustomerPrgHandling.Tool[3].Y:=rSuker3BiasY;
	CustomerPrgHandling.Tool[3].C:=rSuker3PickC;
	//CustomerPrgHandling.Tool[3].Z:=iSuckerHeight;
	CustomerPrgHandling.Tool[4].X:=rSuker4BiasX;
	CustomerPrgHandling.Tool[4].Y:=rSuker4BiasY;
	CustomerPrgHandling.Tool[4].C:=rSuker4PickC;
	//CustomerPrgHandling.Tool[4].Z:=iSuckerHeight;
	
	//保存自动运行参数
	IF xSaveRunPra THEN
		CustomerPrgEdit.SaveRunPra(axSavePrgNo:=p_axSavePrgNo,adr_iCurrentPrgNum:=p_iCurrentPrgNum,xSaveRunPra:=xSaveRunPra,
			rFollowBias_X:=rFollowBias_X,rFollowBias_Y:=rFollowBias_Y,rSuckerDropHeight:=rSuckerDropHeight,
			rBelt1_ClutchPra:=rBelt1_ClutchPra,rBelt2_ClutchPra:=rBelt2_ClutchPra,
			rSuck_Gas_OpenTime:=rSuck_Gas_OpenTime,rBlow_Gas_OpenTime:=rBlow_Gas_OpenTime,rBlowGasTime:=rBlowGasTime,
			iBox_ExceptionDeal:=iBox_ExceptionDeal,
			iSelfadaptPickSwitch:=iSelfadaptPickSwitch,
			rPnPDurationNegativeLimit:=rPnPDurationNegative,
			rPnPDurationPositiveLimit:=rPnPDurationPositive,
			iProdDeformation:=iProdDeformation,
			CustomerPrg:=CustomerPrg,aLRPP_TeachPoints:=aLRPP_TeachPoints);
			
			p_rPnPDurationNegativeLimit:=rPnPDurationNegativeLimit;			
			p_rPnPDurationPositiveLimit:=rPnPDurationPositiveLimit;	
			p_rTorqueForwardControl:=rTorqueForwardControl;	
	END_IF
		
END_IF


//自动运行隐藏主菜单延迟设置	
IF xRunOrStopPrg THEN
	xAutoMenu:=TRUE;
END_IF
DetectStop_Ftrig(CLK:=xRunOrStopPrg, Q=>);
	
IF DetectStop_Ftrig.Q THEN
	fb_TON_Menu.IN:=TRUE;
	fb_TON_Menu.PT:= T#2S; 
END_IF
	
IF fb_TON_Menu.Q=TRUE THEN
	fb_TON_Menu.IN:=FALSE;
	xAutoMenu:=FALSE;
END_IF		
fb_TON_Menu();

//自动运行隐藏主菜单延迟设置	
IF NOT xAutoRun THEN
	iCurrentPrgCmdNum:=1;
	iCommandType:=0;
	iAutoStep:=0;
	xDoNextCmd:=FALSE;
	xChangeMotionType:=TRUE;
	xRunOrStopPrg:=FALSE;
	wstep:=5;       //跳转到待机状态
END_IF
END_ACTION

ACTION A80_SuckBlow:
	
	p_i_Suck1_Num:=	i_Suck1_Num;
	p_i_Blow1_Num:=	i_Blow1_Num;
	//p_iDoShootOut_Num:=iDoShootOut_Num;
	//p_iPrgDoOutputVal_Num:=iPrgDoOutputVal_Num;	
	
	DO_4:=x_Suck1;
END_ACTION

ACTION A60_CameraHandler:
	
IF xMainInit THEN
	// 负荷分配参数
	p_iLoadMode:=iLoadMode;
	p_iRobotNum:=iRobotNum;
	p_iLoadProdNum:=iLoadProdNum;
	p_iLoadDistrRule:=iLoadDistrRule;
	p_arLoadRatio:=arLoadRatio; 
	p_aiServerCommuPort:=aiServerCommuPort;
	p_iSlaveCommuPort:=iSlaveCommuPort;
	
	p_rPallet_DeltaX:=rPallet_DeltaX;
	p_rPallet_DeltaY:=rPallet_DeltaY;	
END_IF
END_ACTION

ACTION A93_SetTorqueLimit:
//**********************************************************************
// Torque limitation
//*************************************************************************

//Get Motor Rated Torque
lrMotorRatedTorque[1]:=L_MC1P_GetRatedTorqueAxis(Axis:=A1 );	
lrMotorRatedTorque[2]:=L_MC1P_GetRatedTorqueAxis(Axis:=A2 );
lrMotorRatedTorque[3]:=L_MC1P_GetRatedTorqueAxis(Axis:=A3 );

//A1
lrTorqueLimit[1]:=lrMotorRatedTorque[1]*A1_TorqueLimitFactor[1];
//A2
lrTorqueLimit[2]:=lrMotorRatedTorque[2]*A2_TorqueLimitFactor[1];
//A3
lrTorqueLimit[3]:=lrMotorRatedTorque[3]*A3_TorqueLimitFactor[1];


fbSetTorqueLimit[1](
	Axis:= A1, 
	xEnable:= xSetTorqueLimitEnable[1],			 
	xSetTorqueLimitPos:=TRUE , 
	lrTorqueLimitPos:=lrTorqueLimit[1], 
	xSetTorqueLimitNeg:=TRUE, 
	lrTorqueLimitNeg:=lrTorqueLimit[1], 
	xBusy=> , 
	xError=> , 
	eErrorID=> );

fbSetTorqueLimit[2](
	Axis:= A2, 
	xEnable:= xSetTorqueLimitEnable[2],
	xSetTorqueLimitPos:=TRUE , 
	lrTorqueLimitPos:=lrTorqueLimit[2], 
	xSetTorqueLimitNeg:=TRUE, 
	lrTorqueLimitNeg:=lrTorqueLimit[2], 
	xBusy=> , 
	xError=> , 
	eErrorID=> );	
	
fbSetTorqueLimit[3](
	Axis:= A3, 
	xEnable:= xSetTorqueLimitEnable[3],
	xSetTorqueLimitPos:=TRUE , 
	lrTorqueLimitPos:=lrTorqueLimit[3], 
	xSetTorqueLimitNeg:=TRUE, 
	lrTorqueLimitNeg:=lrTorqueLimit[3], 
	xBusy=> , 
	xError=> , 
	eErrorID=> );
END_ACTION

ACTION A02_DetectDeviceChoose:
IF iPrdtDetectDevice=Detect_Device.Camera OR  iPrdtDetectDevice=Detect_Device.Computer THEN
	A60_CameraHandler();
END_IF

IF iPrdtDetectDevice=Detect_Device.Sensor THEN
	//A90_SensorHandler();
END_IF
END_ACTION

ACTION A03_PowerCtrl:
//modified in 2016.11.03
Aux1_ABC.xRegulatorOn:=AGBControl.xRegulatorOnALL:=NOT (A1_BrakeDelay.Q OR A2_BrakeDelay.Q OR A3_BrakeDelay.Q OR AuxC_BrakeDelay.Q
								     OR xA1_BrakeOpenStatus OR xA2_BrakeOpenStatus OR xA3_BrakeOpenStatus (*OR wstep=1*));  					
//modified in 2016.11.03									 
IF xTotalConfig AND AGBControl.eAxesGroupState=L_MC4P_AxesGroup_State.GroupDisabled THEN
	Aux1_ABC.xRegulatorOn:=	AGBControl.xRegulatorOnALL:=FALSE;
END_IF		
							 
IF  AGBControl.xRealAxesEnabledALL=TRUE  (*AND wstep<>50*) THEN
	AGBControl.xEnableAxesGroup:=TRUE;		
END_IF

//modified in 2016.11.03
IF xTotalConfig AND NOT xMainInit THEN
	Aux1_ABC.xRegulatorOn:=AGBControl.xEnableAxesGroup:=FALSE;	
END_IF

IF xTotalConfig THEN //一旦进行参数设置STO断开
	AGBControl.xEnableAxesGroup:=FALSE;
END_IF 

fb_TON_STO_Off(IN:=xTotalConfig,pt:=T#2S,Q=>);

IF xTotalConfig THEN //一旦进行参数设置STO断开	
	IF AGBControl.xRegulatorOnALL=FALSE AND fb_TON_STO_Off.Q THEN
		DO_3:=FALSE;
	END_IF	
ELSE	
	DO_3:=TRUE;	
END_IF 

//modified in 2016.11.03	
IF A1.xDriveWarning OR A2.xDriveWarning OR A3.xDriveWarning OR AGBControl.xAxesGroupError OR Aux1_ABC.xError  OR xSystemError THEN
	AGBControl.xRegulatorOnALL:=FALSE;
	AGBControl.xEnableAxesGroup:=FALSE;
	Aux1_ABC.xRegulatorOn:=FALSE;
END_IF 
	//ABC模块上电
//-----------------------------------------------------------------------------/////////////////////////////////////
g_xCameraComOk:=g_xCameraChanelComOk;
// ------------------------------- Systme Conditions ----------------------------------
// Cycle Start Conditions  
g_xCycleReady:= (NOT Delta_Robot.xError) AND (NOT Delta_Robot.xWarning) AND Delta_Robot.xAxesGroupIsHomed
					AND	g_xCameraComOk;
END_ACTION

ACTION A04_ResetFunction:
//modified in 2016.11.03	
Aux1_ABC.xResetError:=AGBControl.xResetAxesGroup:=xResetError ;   //机器人复位
	
IF xResetError=TRUE THEN
	xResetClearBuffer:=TRUE;
	CustomerPrgHandling.xEnable:=FALSE;
	ErrorID:=0;//复位的ErrorID
	WarningID:=0;//复位的WarningID
	iPlaceCounter:=0;
	//LogicControl.xReStart:=TRUE;
ELSE	
	xResetClearBuffer:=FALSE;
	//LogicControl.xReStart:=FALSE;
END_IF
//启动清空 相机或者其它传感器的缓存
ClearBuffer_Rtrig(CLK:=xRunOrStopPrg OR xResetClearBuffer, Q=> );//启动清空相机缓存
LoadDistribution.xClearBuffer:=ClearBuffer_Rtrig.Q;//启动清空相机缓存
BufferHandling.xClearBuffer:=ClearBuffer_Rtrig.Q;//启动清空相机缓存
SensorBufferHandler.xClearBuffer:=ClearBuffer_Rtrig.Q;//启动清空传感器缓存
MultiPickHandling.xClearBuffer:=ClearBuffer_Rtrig.Q;//启动清空相机缓存

CustomerPrgHandling.xPnPReset:=xResetError ;//复位运动模块错误
CustomerPrgHandling.xResetAutoRun:=xResetAutoRun OR xResetError ;//复位自动运行模块错误
END_ACTION

ACTION A40_SetParameters:
IF NOT xAutoRun AND xMainInit THEN
	

	p_iPrdtDetectDevice:=iPrdtDetectDevice; //产品检测装置选择 0：相机；1：传感器；2：上位机通讯指定
	p_rSensorBeltPos:=rSensorBeltPos;	//传感器相对进料带原点的位置
	p_rSensorAuxC:=rSensorAuxC;			//传感器检测产品固定角度   
	
	(*------------------------------------------------机器人及电机参数设置------------------------------------------------------------*)
	IF AGBControl.eAxesGroupState=L_MC4P_AxesGroup_State.GroupDisabled THEN	//AG-disable				
		//在AG.disable下修改X轴的参数
		IF xXaxis_ConfirmPara THEN				  
			//----------启动设置失败定时器------------//
			SetParameter_TON[1].IN:=TRUE;
			SetParameter_TON[1].PT:=T#2S;
			//----------启动设置失败定时器------------//		
			WriteXaxisPara[1].Execute:=TRUE;
			WriteXaxisPara[1].ParameterNumber:=51;
			WriteXaxisPara[1].Value:=rXaxis_PositiveLimit;
			
			WriteXaxisPara[2].Execute:=TRUE;
			WriteXaxisPara[2].ParameterNumber:=52;
			WriteXaxisPara[2].Value:=rXaxis_NegativeLimit;

			IF WriteXaxisPara[1].Done AND WriteXaxisPara[2].Done THEN
				FOR i:=1 TO 2 BY 1 DO
					WriteXaxisPara[i].Execute:=FALSE;
				END_FOR
				xXaxis_ConfirmPara:=FALSE;
				SetParameter_TON[1].IN:=FALSE;//定时器复位
			END_IF	
			
			p_rXaxis_PositiveLimit:=rXaxis_PositiveLimit;
			p_rXaxis_NegativeLimit:=rXaxis_NegativeLimit;
			
		END_IF
		//----------设置失败复位并输出警告信息-----------//
		IF SetParameter_TON[1].Q AND xXaxis_ConfirmPara THEN //如果定时时间到并且设置按钮没有复位,复位并输出报警信息
				SetParameter_TON[1].IN:=FALSE;
				xXaxis_ConfirmPara:=FALSE;
				FOR i:=1 TO 2 BY 1 DO
					WriteXaxisPara[i].Execute:=FALSE;
				END_FOR
				//报警信息
				WarningID:=30051;
		END_IF
		//----------设置失败复位并输出警告信息-----------//
		
			//在AG.disable下修改Y轴的参数
		IF xYaxis_ConfirmPara THEN
			//----------启动设置失败定时器------------//
			SetParameter_TON[2].IN:=TRUE;
			SetParameter_TON[2].PT:=T#2S;
			//----------启动设置失败定时器------------//
		
			WriteYaxisPara[1].Execute:=TRUE;
			WriteYaxisPara[1].ParameterNumber:=51;
			WriteYaxisPara[1].Value:=rYaxis_PositiveLimit;
			
			WriteYaxisPara[2].Execute:=TRUE;
			WriteYaxisPara[2].ParameterNumber:=52;
			WriteYaxisPara[2].Value:=rYaxis_NegativeLimit;						
			
			IF WriteYaxisPara[1].Done AND WriteYaxisPara[2].Done THEN
				FOR i:=1 TO 2 BY 1 DO
					WriteYaxisPara[i].Execute:=FALSE;
				END_FOR
				xYaxis_ConfirmPara:=FALSE;
				SetParameter_TON[2].IN:=FALSE;//定时器复位
			END_IF									
			p_rYaxis_PositiveLimit:=rYaxis_PositiveLimit;
			p_rYaxis_NegativeLimit:=rYaxis_NegativeLimit;
		END_IF
		//----------设置失败复位并输出警告信息-----------//
		IF SetParameter_TON[2].Q AND xYaxis_ConfirmPara THEN //如果定时时间到并且设置按钮没有复位,复位并输出报警信息
			SetParameter_TON[2].IN:=FALSE;
			xYaxis_ConfirmPara:=FALSE;
			FOR i:=1 TO 2 BY 1 DO
				WriteYaxisPara[i].Execute:=FALSE;
			END_FOR
			//报警信息
			WarningID:=30052;
		END_IF
		//----------设置失败复位并输出警告信息-----------//	
		

			//在AG.disable下修改Z轴的参数
		IF xZaxis_ConfirmPara THEN
			//----------启动设置失败定时器------------//
			SetParameter_TON[3].IN:=TRUE;
			SetParameter_TON[3].PT:=T#2S;
			//----------启动设置失败定时器------------//
			
			WriteZaxisPara[1].Execute:=TRUE;
			WriteZaxisPara[1].ParameterNumber:=51;
			WriteZaxisPara[1].Value:=rZaxis_PositiveLimit;
			
			WriteZaxisPara[2].Execute:=TRUE;
			WriteZaxisPara[2].ParameterNumber:=52;
			WriteZaxisPara[2].Value:=rZaxis_NegativeLimit;
						
			
			IF WriteZaxisPara[1].Done AND WriteZaxisPara[2].Done   THEN
				FOR i:=1 TO 2 BY 1 DO
					WriteZaxisPara[i].Execute:=FALSE;
				END_FOR
				xZaxis_ConfirmPara:=FALSE;
				SetParameter_TON[3].IN:=FALSE;//定时器复位
			END_IF	
						                                
			p_rZaxis_PositiveLimit:=rZaxis_PositiveLimit;
			p_rZaxis_NegativeLimit:=rZaxis_NegativeLimit;	
		END_IF
		//----------设置失败复位并输出警告信息-----------//
		IF SetParameter_TON[3].Q AND xZaxis_ConfirmPara THEN //如果定时时间到并且设置按钮没有复位,复位并输出报警信息
			SetParameter_TON[3].IN:=FALSE;
			xZaxis_ConfirmPara:=FALSE;
			FOR i:=1 TO 2 BY 1 DO
				WriteZaxisPara[i].Execute:=FALSE;
			END_FOR
			//报警信息
			WarningID:=30053;
		END_IF
		//----------设置失败复位并输出警告信息-----------//	
		
		//在AG.disable下修改A1轴的参数
		IF xA1_ConfirmPara THEN
			//----------启动设置失败定时器------------//
			SetParameter_TON[4].IN:=TRUE;
			SetParameter_TON[4].PT:=T#2S;
			//----------启动设置失败定时器------------//
			CASE WriteA1_Step OF
			0:
				WriteA1axisPara[1].Execute:=TRUE;
				WriteA1axisPara[1].ParameterNumber:=51;
				WriteA1axisPara[1].Value:=rA1_PositiveLimit;
				IF WriteA1axisPara[1].Done THEN				
					WriteA1axisPara[1].Execute:=FALSE;
					WriteA1_Step:=1;
				END_IF
			1:
				WriteA1axisPara[1].Execute:=TRUE;
				WriteA1axisPara[1].ParameterNumber:=52;
				WriteA1axisPara[1].Value:=rA1_NegativeLimit;
				IF WriteA1axisPara[1].Done THEN				
					WriteA1axisPara[1].Execute:=FALSE;
					WriteA1_Step:=2;
				END_IF
			2:
				WriteA1axisPara[1].Execute:=TRUE;
				WriteA1axisPara[1].ParameterNumber:=L_MC1P_IndexToParameter(16#2900,1,4);
				WriteA1axisPara[1].Value:=rA1_Vel_P1*100000;
				IF WriteA1axisPara[1].Done THEN				
					WriteA1axisPara[1].Execute:=FALSE;
					WriteA1_Step:=3;
				END_IF
			3:
				WriteA1axisPara[1].Execute:=TRUE;
				WriteA1axisPara[1].ParameterNumber:=L_MC1P_IndexToParameter(16#2900,2,2);
				WriteA1axisPara[1].Value:=rA1_Vel_I1*10;
				IF WriteA1axisPara[1].Done THEN				
					WriteA1axisPara[1].Execute:=FALSE;
					WriteA1_Step:=4;
				END_IF
			
			4:
				WriteA1axisPara[1].Execute:=TRUE;
				WriteA1axisPara[1].ParameterNumber:=L_MC1P_IndexToParameter(16#2980,0,4);
				WriteA1axisPara[1].Value:=rA1_Pos_P1*100;
				IF WriteA1axisPara[1].Done THEN				
					WriteA1axisPara[1].Execute:=FALSE;
					WriteA1_Step:=0;
					xA1_ConfirmPara:=FALSE; //确定按钮复位
					SetParameter_TON[4].IN:=FALSE; //定时器复位
				END_IF
			END_CASE
			
			
			p_rA1_PositiveLimit:=rA1_PositiveLimit	;
			p_rA1_NegativeLimit:=rA1_NegativeLimit	;
			p_rA1_Vel_P1      :=rA1_Vel_P1 ;		 
			p_rA1_Vel_I1      :=rA1_Vel_I1	;	 
			p_rA1_Pos_P1	  :=rA1_Pos_P1;
		END_IF
		//----------设置失败复位并输出警告信息-----------//
		IF SetParameter_TON[4].Q AND xA1_ConfirmPara THEN //如果定时时间到并且设置按钮没有复位,复位并输出报警信息
				SetParameter_TON[4].IN:=FALSE;
				xA1_ConfirmPara:=FALSE;//确定按钮复位
				WriteA1axisPara[1].Execute:=FALSE;
				WriteA1_Step:=0;//步骤归零
				//报警信息
				WarningID:=30054;
		END_IF
		//----------设置失败复位并输出警告信息-----------//	
				
		//在AG.disable下修改A2轴的参数
		IF xA2_ConfirmPara THEN		
			//----------启动设置失败定时器------------//
			SetParameter_TON[5].IN:=TRUE;
			SetParameter_TON[5].PT:=T#2S;
			//----------启动设置失败定时器------------//
			CASE WriteA2_Step OF
				0:
					WriteA2axisPara[1].Execute:=TRUE;
					WriteA2axisPara[1].ParameterNumber:=51;
					WriteA2axisPara[1].Value:=rA2_PositiveLimit;
					IF WriteA2axisPara[1].Done THEN				
						WriteA2axisPara[1].Execute:=FALSE;
						WriteA2_Step:=1;
					END_IF
				1:
					WriteA2axisPara[1].Execute:=TRUE;
					WriteA2axisPara[1].ParameterNumber:=52;
					WriteA2axisPara[1].Value:=rA2_NegativeLimit;
					IF WriteA2axisPara[1].Done THEN				
						WriteA2axisPara[1].Execute:=FALSE;
						WriteA2_Step:=2;
					END_IF
				2:
					WriteA2axisPara[1].Execute:=TRUE;
					WriteA2axisPara[1].ParameterNumber:=L_MC1P_IndexToParameter(16#3100,1,4);
					WriteA2axisPara[1].Value:=rA2_Vel_P2*100000;
					IF WriteA2axisPara[1].Done THEN				
						WriteA2axisPara[1].Execute:=FALSE;
						WriteA2_Step:=3;
					END_IF
				3:
					WriteA2axisPara[1].Execute:=TRUE;
					WriteA2axisPara[1].ParameterNumber:=L_MC1P_IndexToParameter(16#3100,2,2);
					WriteA2axisPara[1].Value:=rA2_Vel_I2*10;
					IF WriteA2axisPara[1].Done THEN				
						WriteA2axisPara[1].Execute:=FALSE;
						WriteA2_Step:=4;
					END_IF
				
				4:
					WriteA2axisPara[1].Execute:=TRUE;
					WriteA2axisPara[1].ParameterNumber:=L_MC1P_IndexToParameter(16#3180,0,4);
					WriteA2axisPara[1].Value:=rA2_Pos_P2*100;
					IF WriteA2axisPara[1].Done THEN				
						WriteA2axisPara[1].Execute:=FALSE;
						WriteA2_Step:=0;
						xA2_ConfirmPara:=FALSE; //确定按钮复位
						SetParameter_TON[5].IN:=FALSE; //定时器复位
					END_IF
			END_CASE
				
			p_rA2_PositiveLimit:=	rA2_PositiveLimit;
			p_rA2_NegativeLimit:=	rA2_NegativeLimit;
			p_rA2_Vel_P2	   :=	rA2_Vel_P2;      
			p_rA2_Vel_I2	   :=	rA2_Vel_I2;      
			p_rA2_Pos_P2	   :=   rA2_Pos_P2;
		END_IF
		//----------设置失败复位并输出警告信息-----------//
		IF SetParameter_TON[5].Q AND xA2_ConfirmPara THEN //如果定时时间到并且设置按钮没有复位,复位并输出报警信息
				SetParameter_TON[5].IN:=FALSE;
				xA2_ConfirmPara:=FALSE;
				WriteA2axisPara[1].Execute:=FALSE;
				WriteA2_Step:=0;//步骤归零
				//报警信息
				WarningID:=30055;
		END_IF
		//----------设置失败复位并输出警告信息-----------//	
	
		//在AG.disable下修改A3轴的参数
		IF xA3_ConfirmPara THEN		
			//----------启动设置失败定时器------------//
			SetParameter_TON[6].IN:=TRUE;
			SetParameter_TON[6].PT:=T#2S;
			//----------启动设置失败定时器------------//
			CASE WriteA3_Step OF
				0:
					WriteA3axisPara[1].Execute:=TRUE;
					WriteA3axisPara[1].ParameterNumber:=51;
					WriteA3axisPara[1].Value:=rA3_PositiveLimit;
					IF WriteA3axisPara[1].Done THEN				
						WriteA3axisPara[1].Execute:=FALSE;
						WriteA3_Step:=1;
					END_IF
				1:
					WriteA3axisPara[1].Execute:=TRUE;
					WriteA3axisPara[1].ParameterNumber:=52;
					WriteA3axisPara[1].Value:=rA3_NegativeLimit;
					IF WriteA3axisPara[1].Done THEN				
						WriteA3axisPara[1].Execute:=FALSE;
						WriteA3_Step:=2;
					END_IF
				2:
					WriteA3axisPara[1].Execute:=TRUE;
					WriteA3axisPara[1].ParameterNumber:=L_MC1P_IndexToParameter(16#2900,1,4);
					WriteA3axisPara[1].Value:=rA3_Vel_P3*100000;
					IF WriteA3axisPara[1].Done THEN				
						WriteA3axisPara[1].Execute:=FALSE;
						WriteA3_Step:=3;
					END_IF
				3:
					WriteA3axisPara[1].Execute:=TRUE;
					WriteA3axisPara[1].ParameterNumber:=L_MC1P_IndexToParameter(16#2900,2,2);
					WriteA3axisPara[1].Value:=rA3_Vel_I3*10;
					IF WriteA3axisPara[1].Done THEN				
						WriteA3axisPara[1].Execute:=FALSE;
						WriteA3_Step:=4;
					END_IF
				
				4:
					WriteA3axisPara[1].Execute:=TRUE;
					WriteA3axisPara[1].ParameterNumber:=L_MC1P_IndexToParameter(16#2980,0,4);
					WriteA3axisPara[1].Value:=rA3_Pos_P3*100;
					IF WriteA3axisPara[1].Done THEN				
						WriteA3axisPara[1].Execute:=FALSE;
						WriteA3_Step:=0;
						xA3_ConfirmPara:=FALSE; //确定按钮复位
						SetParameter_TON[6].IN:=FALSE; //定时器复位
					END_IF
			END_CASE

			p_rA3_PositiveLimit	 :=	rA3_PositiveLimit;
			p_rA3_NegativeLimit  :=	rA3_NegativeLimit;
			p_rA3_Vel_P3		 :=	rA3_Vel_P3;      
			p_rA3_Vel_I3	 	 :=	rA3_Vel_I3;      
			p_rA3_Pos_P3	  	 := rA3_Pos_P3;
			
		END_IF
		//----------设置失败复位并输出警告信息-----------//
		IF SetParameter_TON[6].Q AND xA3_ConfirmPara THEN //如果定时时间到并且设置按钮没有复位,复位并输出报警信息
				SetParameter_TON[6].IN:=FALSE;
				xA3_ConfirmPara:=FALSE;
				WriteA3axisPara[1].Execute:=FALSE;
				WriteA3_Step:=0;//步骤归零
				//报警信息
				WarningID:=30056;
		END_IF
		//----------设置失败复位并输出警告信息-----------//	
	
		//在AG.disable下修改AuxC轴的参数
		IF xAuxC_ConfirmPara THEN		
			//----------启动设置失败定时器------------//
			SetParameter_TON[7].IN:=TRUE;
			SetParameter_TON[7].PT:=T#3S;
			//----------启动设置失败定时器------------//
			CASE WriteAuxC_Step OF
				0:
					WriteAuxCaxisPara[1].Execute:=TRUE;
					WriteAuxCaxisPara[1].ParameterNumber:=51;
					WriteAuxCaxisPara[1].Value:=rAuxC_PositiveLimit;
					IF WriteAuxCaxisPara[1].Done THEN				
						WriteAuxCaxisPara[1].Execute:=FALSE;
						WriteAuxC_Step:=1;
					END_IF
				1:
					WriteAuxCaxisPara[1].Execute:=TRUE;
					WriteAuxCaxisPara[1].ParameterNumber:=52;
					WriteAuxCaxisPara[1].Value:=rAuxC_NegativeLimit;
					IF WriteAuxCaxisPara[1].Done THEN				
						WriteAuxCaxisPara[1].Execute:=FALSE;
						WriteAuxC_Step:=2;
					END_IF
				2:
					WriteAuxCaxisPara[1].Execute:=TRUE;
					WriteAuxCaxisPara[1].ParameterNumber:=L_MC1P_IndexToParameter(16#3100,1,4);
					WriteAuxCaxisPara[1].Value:=rAuxC_Vel_P3*100000;
					IF WriteAuxCaxisPara[1].Done THEN				
						WriteAuxCaxisPara[1].Execute:=FALSE;
						WriteAuxC_Step:=3;
					END_IF
				3:
					WriteAuxCaxisPara[1].Execute:=TRUE;
					WriteAuxCaxisPara[1].ParameterNumber:=L_MC1P_IndexToParameter(16#3100,2,2);
					WriteAuxCaxisPara[1].Value:=rAuxC_Vel_I3*10;
					IF WriteAuxCaxisPara[1].Done THEN				
						WriteAuxCaxisPara[1].Execute:=FALSE;
						WriteAuxC_Step:=4;
					END_IF
				
				4:
					WriteAuxCaxisPara[1].Execute:=TRUE;
					WriteAuxCaxisPara[1].ParameterNumber:=L_MC1P_IndexToParameter(16#3180,0,4);
					WriteAuxCaxisPara[1].Value:=rAuxC_Pos_P3*100;
					IF WriteAuxCaxisPara[1].Done THEN				
						WriteAuxCaxisPara[1].Execute:=FALSE;
						WriteAuxC_Step:=0;
						xAuxC_ConfirmPara:=FALSE; //确定按钮复位
						SetParameter_TON[7].IN:=FALSE; //定时器复位
					END_IF
			END_CASE
		
			
			p_rAuxC_PositiveLimit	:=rAuxC_PositiveLimit;	
			p_rAuxC_NegativeLimit	:=rAuxC_NegativeLimit;	
			p_rAuxC_Vel_P3			:=rAuxC_Vel_P3	;		
			p_rAuxC_Vel_I3			:=rAuxC_Vel_I3	;		
			p_rAuxC_Pos_P3			:=rAuxC_Pos_P3	;		
		END_IF
		
		//----------设置失败复位并输出警告信息-----------//
		IF SetParameter_TON[7].Q AND xAuxC_ConfirmPara THEN //如果定时时间到并且设置按钮没有复位,复位并输出报警信息
				SetParameter_TON[7].IN:=FALSE;
				xAuxC_ConfirmPara:=FALSE;
				WriteAuxCaxisPara[1].Execute:=FALSE;
				WriteAuxC_Step:=0;//步骤归零
				//报警信息
				WarningID:=30057;
		END_IF
		//----------设置失败复位并输出警告信息-----------//	
	
		//在AG.disable下修改Infeeder轴的参数
		IF xInfeederConfirmParameter THEN
			//InFeedPower.Enable:=FALSE;
			 //----------启动设置失败定时器------------//
				SetParameter_TON[8].IN:=TRUE;
				SetParameter_TON[8].PT:=T#2S;
				//----------启动设置失败定时器------------//
			// IF Infeeder.eAxisState=L_MC1P_AXIS_State.Disabled THEN

				ChangeInfeederPara.xExecute:=TRUE;				
				ChangeInfeederPara.xOrientation:=xInfeederDirection;
				ChangeInfeederPara.xSetOrientation:=TRUE;
				
				//ChangeInfeederPara.dwPosResolution:=4096;//REAL_TO_DWORD(rInfeederPosResolution);
				//ChangeInfeederPara.xSetPosResolution:=TRUE;
				
				ChangeInfeederPara.eTraversingRange:=L_MC1P_TraversingRange.Modulo;
				ChangeInfeederPara.xSetTraversingRange:=TRUE;
				
				ChangeInfeederPara.dwGearNumerator:=REAL_TO_DWORD(rInfeederGearRedRatio*1000*rInfeederPosResolution/2048);
				ChangeInfeederPara.dwGearDenominator:=REAL_TO_DWORD(1000);	
				ChangeInfeederPara.xSetGearFactor:=TRUE;
				
				ChangeInfeederPara.lrFeedconstant:=rInfeederFeedConst;			
				ChangeInfeederPara.xSetFeedconstant:=TRUE;
				
				//ChangeInfeederPara.lrCycleLength:=rInfeederCycleLength;
				//ChangeInfeederPara.xSetCycleLength:=TRUE;
				
				IF ChangeInfeederPara.xDone  THEN

					ChangeInfeederPara.xExecute:=FALSE;
					xInfeederConfirmParameter:=FALSE;
					SetParameter_TON[8].IN:=FALSE; //定时器复位
				END_IF
				
				p_xInfeederDirection		:=xInfeederDirection		;
				p_rInfeederPosResolution    :=rInfeederPosResolution    ;
				p_rInfeederGearRedRatio	    :=rInfeederGearRedRatio	    ;
				p_rInfeederFeedConst	    :=rInfeederFeedConst	    ;
				//p_rInfeederCycleLength	    :=rInfeederCycleLength	    ;
			//END_IF						
		END_IF
				
		//----------设置失败复位并输出警告信息-----------//
		IF SetParameter_TON[8].Q AND xInfeederConfirmParameter THEN //如果定时时间到并且设置按钮没有复位,复位并输出报警信息
			
				SetParameter_TON[8].IN:=FALSE;
				xInfeederConfirmParameter:=FALSE;
				ChangeInfeederPara.xExecute:=FALSE;
				//InFeedPower.Enable:=TRUE;//恢复使能
				//报警信息
				WarningID:=30058;
		END_IF
		//----------设置失败复位并输出警告信息-----------//	
		
		//在AG.disable下修改Outfeeder轴的参数
		IF xOutfeederConfirmParameter THEN
			// OutFeedPower.Enable:=FALSE;
				//----------启动设置失败定时器------------//
				SetParameter_TON[9].IN:=TRUE;
				SetParameter_TON[9].PT:=T#2S;
				//----------启动设置失败定时器------------//
			// IF Outfeeder.eAxisState=L_MC1P_AXIS_State.Disabled THEN
	
				ChangeOutfeederPara.xExecute:=TRUE;		
				ChangeOutfeederPara.xOrientation:=xOutfeederDirection;
				ChangeOutfeederPara.xSetOrientation:=TRUE;
								
				//ChangeOutfeederPara.dwPosResolution:=UINT_TO_DWORD(rOutfeederPosResolution);
				//ChangeOutfeederPara.xSetPosResolution:=TRUE;
				
				ChangeOutfeederPara.dwGearNumerator:=REAL_TO_DWORD(rOutfeederGearRedRatio*1000*rOutfeederPosResolution/2048);
				ChangeOutfeederPara.dwGearDenominator:=REAL_TO_DWORD(1000);	
				ChangeOutfeederPara.xSetGearFactor:=TRUE;
				
				ChangeOutfeederPara.lrFeedconstant:=rOutfeederFeedConst;			
				ChangeOutfeederPara.xSetFeedconstant:=TRUE;
				
				//ChangeOutfeederPara.lrCycleLength:=rOutfeederCycleLength;
				//ChangeOutfeederPara.xSetCycleLength:=TRUE; 
				
				IF ChangeOutfeederPara.xDone THEN
					ChangeOutfeederPara.xExecute:=FALSE;
					xOutfeederConfirmParameter:=FALSE;
					SetParameter_TON[9].IN:=FALSE; //定时器复位
					//OutFeedPower.Enable:=TRUE;//恢复使能
				END_IF
				
				p_xOutfeederDirection		:=xOutfeederDirection		;
				p_rOutfeederPosResolution	:=rOutfeederPosResolution   ;
				p_rOutfeederGearRedRatio	:=rOutfeederGearRedRatio	;
				p_rOutfeederFeedConst		:=rOutfeederFeedConst		;
				//p_rOutfeederCycleLength	    :=rOutfeederCycleLength	    ;
			//END_IF			
		END_IF
		//----------设置失败复位并输出警告信息-----------//
		IF SetParameter_TON[9].Q AND xOutfeederConfirmParameter THEN //如果定时时间到并且设置按钮没有复位,复位并输出报警信息
				SetParameter_TON[9].IN:=FALSE;
				xOutfeederConfirmParameter:=FALSE;
				ChangeOutfeederPara.xExecute:=FALSE;
				//OutFeedPower.Enable:=TRUE;//恢复使能
				//报警信息
				WarningID:=30059;
		END_IF
		//----------设置失败复位并输出警告信息-----------//	
		
	END_IF						
END_IF


	WriteXaxisPara[1](Axis:=Axis_X); WriteXaxisPara[2](Axis:=Axis_X);	
	WriteYaxisPara[1](Axis:=Axis_Y); WriteYaxisPara[2](Axis:=Axis_Y);		
	WriteZaxisPara[1](Axis:=Axis_Z); WriteZaxisPara[2](Axis:=Axis_Z);
	WriteA1axisPara[1](Axis:=A1); 	
	WriteA2axisPara[1](Axis:=A2); 
	WriteA3axisPara[1](Axis:=A3); 
	//WriteAuxCaxisPara[1](Axis:=AxisYaw);
	//ChangeInfeederPara(Axis:=Infeeder);
	//ChangeOutfeederPara(Axis:=Outfeeder);
	
	SetParameter_TON[1]();SetParameter_TON[2]();SetParameter_TON[3]();SetParameter_TON[4]();SetParameter_TON[5]();
	SetParameter_TON[6]();SetParameter_TON[7]();SetParameter_TON[8]();SetParameter_TON[9]();
END_ACTION

ACTION A94_RealAxisFilter:

L_MC1P_AverageFilterSetValues_A1(
	Axis:= A1,
	xEnable:= xFilterEnable,
	eExecutionIndex:= 1,
	xIgnoreFilterOnStop := FALSE,
	xBusy=> ,
	xActive=> ,
	xError=> ,
	eErrorID=> ,
	lrSetPosOut=> ,
	lrSetVelOut=> ,
	lrSetAccOut=> ,
	lrSetTorqueOut=> ,
	wFilterDepth:= wFilterDepth);

L_MC1P_AverageFilterSetValues_A2(
	Axis:= A2,
	xEnable:= xFilterEnable,
	eExecutionIndex:= 1,
	xIgnoreFilterOnStop:= FALSE,
	xBusy=> ,
	xActive=> ,
	xError=> ,
	eErrorID=> ,
	lrSetPosOut=> ,
	lrSetVelOut=> ,
	lrSetAccOut=> ,
	lrSetTorqueOut=> ,
	wFilterDepth:= wFilterDepth);

L_MC1P_AverageFilterSetValues_A3(
	Axis:= A3,
	xEnable:= xFilterEnable,
	eExecutionIndex:= 1,
	xIgnoreFilterOnStop := FALSE,
	xBusy=> ,
	xActive=> ,
	xError=> ,
	eErrorID=> ,
	lrSetPosOut=> ,
	lrSetVelOut=> ,
	lrSetAccOut=> ,
	lrSetTorqueOut=> ,
	wFilterDepth:= wFilterDepth);
END_ACTION

ACTION A96_IK:

//**********************************************************************
// INVERSE KINEMATICS
//**********************************************************************
fb_InverseKinematics(
	a:= 170.0/1000.0, 
	b:= SQRT(71.42*71.42-50.0*50.0)/1000.0, 
	L1:= 450.0/1000.0, 
	L2:= 1000.0/1000.0, 
	x:= Axis_X.lrSetPosition/1000.0, 
	y:= -Axis_Y.lrSetPosition/1000.0, 
	z:= -Axis_Z.lrSetPosition/1000.0, 
	theta1=> , 
	theta2=> , 
	theta3=> );
END_ACTION

ACTION A98_TFFControl:
//**********************************************************************
//Torque Feedforward control
//**********************************************************************
lrRatioOfTorqueFeedForward:=REAL_TO_LREAL(rTorqueForwardControl);	
LCP_MC4P_TorqueComputation_1(
	AxesGroup:= Delta_Robot,
	xEnable:=(lrRatioOfTorqueFeedForward>0.0)AND xAutoRun,	
	xFeedforwardControlEnable:= (lrRatioOfTorqueFeedForward>0.0)AND xAutoRun,//xFeedforwardControl, 
	lrRatioOfTorqueOffset:= lrRatioOfTorqueFeedForward, 
	lrMassOfProximalLink:= 2.182, 
	lrMassOfDistalLink:= 1.138, 
	lrMassOfMovingPlatform:= 0.663, 
	lrInertiaOfMotorAndGearbox:=(2.17+0.56), 
	xFrictionCompeEnable:= xFrictionCompe, 
	alrCoulombFriction:= alrCoulombFriction, 
	alrViscousFriction:= alrViscousFriction,
	alrComputedTorque=> , 
	alrFrictionComp=> , 
	alrSetTorqueOut=> );
END_ACTION

END_PROGRAM

// Controller_3200C/Application/CustomerPrgHandling
PROGRAM CustomerPrgHandling
VAR_IN_OUT	
	xRunOrStopPrg						: BOOL;			//启动
	Delta_Robot							: AXES_GROUP_KIN; //运动学模型
	AuxC								: AXIS_REF;		//旋转轴
	Infeeder							: AXIS_REF;		//进料带
	Outfeeder							: AXIS_REF; 		//出料带
	xMasterOutfeederStart				: BOOL;			//主机出料带启动信号
	xSlaveOutfeederStart				: BOOL;			//从机出料带启动信号
	iOutputVal							: BOOL;			//外部输出信号
	ErrorID								: UINT;			//错误ID
END_VAR
VAR_INPUT
	DI_5								:BOOL;						//对外开放
	DI_6								:BOOL;						//对外开放
	DI_7								:BOOL;						//对外开放	
	xRunInter							:BOOL;						//启动
	xStopInter							:BOOL;						//停止
	xEnable								:BOOL;						//使能
	xResetAutoRun						:BOOL;						//复位
	xProdInfoReady						:BOOL;						//产品准备信号
	xProdInfoFirstReady					:BOOL;						//产品过最小抓取线准备信号
	xProdInfoNextReady					:BOOL;
	xOutFeedStart						:BOOL;						//最后一抓箱体启动信号
	CustomerPrg							:L_RPP_CustomerProgram;		//用户程序
	sInFeedBeltOrigin					:BeltOrigin;				//进料带原点
	sOutFeedBeltOrigin					:BeltOrigin;				//出料带原点
	lrInfeedDeltaX						:LREAL;						//进料带产品位置-X
	lrInfeedDeltaY						:LREAL;						//进料带产品位置-Y
	rFollowBias_X						:REAL;	// 1 抓取位置微调-X
	rFollowBias_Y						:REAL;	// 2 抓取位置微调-Y
	rSuckerDropHeight					:REAL;  // 3 抓取位置微调-Z
	rInfeedClutchPra					:REAL;  // 4 进料带跟踪系数
	rOutfeedClutchPra					:REAL;  // 5 出料带跟踪系数
	rBlowOpenTime						:REAL;	// 6 吸盘提前吹气时间 ms
	rSuckOpenTime						:REAL;	// 7 吸盘提前吸气时间 ms
	rBlowGasTime						:REAL;  // 8 吸盘吹气持续时间 ms
	iBox_ExceptionDeal					:INT;   // 9 装箱异常处理 0、1
	iSelfadaptPickSwitch				:INT;   //10 启动变节拍自适应抓取
	rPnPDurationNegativeLimit			:REAL;	//   12运动时间下限					
 	rPnPDurationPositiveLimit			:REAL;	//   13运动时间上限				
	
	iProdDeformation					:INT;   //11 产品变形量	
	xPnPReset							:BOOL;	// PnP模块复位
	lrPosAuxC							:LREAL;	// 相机拍摄的产品角度
	lrNextProdAuxC						:LREAL; //下一个产品的角度
	lrCurrentAuxC						:LREAL; // 当前辅助轴位置
	//lrOutfeedCameraDeltaX				:LREAL;	
	//lrOutfeedCameraDeltaY				:LREAL;
	rProductAdd_Z						:REAL;	// 产品高度 h	
	//xCameraCycleReady					:BOOL;	// 自动抓取就绪信号
	xDetectBoxSwitch					:BOOL;  // 检测箱体光电开关
	rBoxLength							:REAL;  // 箱体长度
	rBoxBiasLength						:REAL;  // 箱体偏置长度
	iBoxInterval						:INT;	// 检测箱体间隔
	Tool								:ARRAY[1..4] OF SuckerInfo;//吸盘
	iNewProdNum							:INT;	//检测物体需要的外部触发信号数量
	rBoxOutfeederVel					:REAL;	// 装箱时出料带的速度
	rBoxPickTime						:REAL;  // 装箱抓取物料时间
	rBoxPlaceTime 						:REAL;  // 装箱放置物料时间
	rBoxDetectPosX						:REAL;  // 装箱检测箱体的初始位置
	
	//*************************************************
	rCoefMaxOfStartAndEndR				: ARRAY[1..2] OF REAL;						
	iAux1ExePointPassed					: ARRAY[1..2] OF INT;							
	rAux1DurationRatio					: ARRAY[1..2] OF REAL;								
	iAux1MotionLaw						: ARRAY[1..2] OF INT;	//2: 5th ploy; 3: 7th ploy						
	rStartAlphaRatio					: ARRAY[1..2,1..3] OF REAL;						
	rEndAlphaRatio						: ARRAY[1..2,7..9] OF REAL;
		
	//2017.03.30	
	lrDistToMinCapLForCycleAdaptive		: LREAL;
	lrMinCaptureLine					: LREAL;
	lrMaxCaptureLine					: LREAL;	
	xBoxEnable							: BOOL:=TRUE;
	rPalletPickDeltaX					: REAL; //Pick托盘的x向间距 2017.12.13
	rPalletPickDeltaY					: REAL; //Pick托盘的y向间距 2017.12.13
	rPalletPlaceDeltaX					: REAL; //Place托盘的x向间距2017.12.13
	rPalletPlaceDeltaY					: REAL; //Place托盘的y向间距2017.12.13
END_VAR
		
VAR_OUTPUT
	xBoxFull							:BOOL; //装箱是否装满
	xBoxMoveEnable						:BOOL:=TRUE; //判断启动时刻，箱体是否可以移动
	iCommandType						:INT;	//当前程序类型
	iCurrentPrgCmdNum					:INT;	//当前程序运行行号
	xFirstProdDel		 				:BOOL;  //删除第一个产品信息
	lrPaPDuration		    			:LREAL; //抓取时间
	xSuck								:BOOL;	//吸气
	xSuck2								:BOOL;	//吸气2
	xBlow								:BOOL;	//吹气
	xWarning							:BOOL;	//警告
	iPickedPrdNr						:INT;	//已抓取产品数量
	iActiveToolNr						:INT;  //多抓-已激活工具编号
END_VAR
VAR
	xRunPermission						: BOOL;
	iCommandIndex						: INT;	//指令索引
	g_lrCameraInitialPos				: LREAL;	// 相机拍摄到的物体初始值
	g_lrTargetAngle						: LREAL;				// 辅助旋转轴角度  单位: 度
	g_lrAuxCLayDonwTarPos				: LREAL;	// 辅助旋转轴角度  单位: 度
	PlaceBelt_Pos						: CoordTransPos;
	fb_P2P								: MC_MoveDirectAbsolute;
	fb_MoveLinear						: MC_MoveLinearAbsolute;
	fb_MoveCircle						: MC_MoveCircularAbsolute;
	MC_TrackConveyorBelt_U				: ARRAY [1..10] OF MC_TrackConveyorBelt;
	MC_TrackConveyorBelt_U1				: MC_TrackConveyorBelt;				
	MC_TrackConveyorBelt_U1_PCS_7		: MC_TrackConveyorBelt;	
	MC_TrackConveyorBelt_U1_PCS_8		: MC_TrackConveyorBelt;	
	MC_TrackConveyorBelt_U1_PCS_9		: MC_TrackConveyorBelt;				
	MC_TrackConveyorBelt_U2				: MC_TrackConveyorBelt;				
	TrackingCorrectAxisStateBeltIn		: TrackingCorrectAxisState;
	TrackingCorrectAxisStateBeltOut		: TrackingCorrectAxisState;	
	L_RPP_PickPlace_0					: L_RPP_PickPlace;
	L_RPP_PickPlace_1					: L_RPP_PickPlace;							
	//L_RPP_PickPlace_2					: L_RPP_PickPlace;							
	MoveToWaitPoint0					: MoveToWaitPoint;						
	Robot_Stop							: MC_GroupStop;						
	AuxC_Stop							: MC_Stop;											
	Ac_CaptureTarget					: AuxC_CaptureTarget;
	Ac_LayDownTarget					: AuxC_LayDownTarget;

	Pick0_RTrig							: R_TRIG;
	Pick1_RTrig							: R_TRIG;
	Run_RTrig							: R_TRIG;
	Stop_RTrig							: R_TRIG;
    fb_TON								: TON;
	fb_TON3								: TON;
	fb_TON_Dur1							: TON;
	fb_TON_Delay						: TON;
	fb_TON_ResetPnP						: TON;
	TOF_PrDel							: TOF;
	TOF_BoxFull							:TOF;
	//xNew_Place						:BOOL;
	//iPrDel_Cnt						:INT;
	//ProDel_Rtrig						:R_TRIG;
	xSuckInter							:BOOL;
	xSuckInter2							:BOOL;
	xBlowInter							:BOOL;
	iSuckDiscNr							:INT;
	xSuckBlowLock						:BOOL;
	t_waitime							:TIME; 		//ms
	xChangeMotionType					:BOOL:=TRUE;
	iAutoStep							:INT;
	xDoNextCmd							:BOOL; 		//
	xSearchPlaceCmd						:BOOL;
	iJpCnt								:INT;
	iJumpPlaceNo						:INT;//第一个Place指令的行号
	iJumpNum							:INT;//跳转行号
	iJumpTimes							:INT;//跳转次数
	iJumpCount							:INT;//跳转计数变量
	aiJumpCount							:ARRAY [1..50] OF INT;
	iJumpOutInEvent						:INT;	//定义内部跳出条件
	xJumpEndCondition					:BOOL;	//定义跳出条件
	iPreJumpPrgNum						:INT;	//跳转前的程序行
	iExtWaitEventNum					:INT;	//等待外部事件号
	iInterWaitEventNum					:INT;	//等待内部事件号
	iInterEventJumpNo					:INT;	//等待内部跳转行号
	rMinPlaceLine						:REAL;
	rMaxPlaceLine						:REAL;
	rMinPickLine						:REAL;
	rMaxPickLine						:REAL;

	//iOutputNo							:INT;
	wPickAloneStep:						WORD;		
	wPickWithBeltStep:					WORD;		
	wPlaceAloneStep:					WORD;		
	wPlaceWithBeltStep:					WORD;			
	wPlaceSafeStep:						WORD;		
	AuxMode: 							ARRAY[1..6] OF L_MC4P_AuxMode:= [0,0,0,0,0,0];			
	iOutputDuration						:INT;
	iInputSignalNo  					:INT;
	xInputSetValue						:BOOL;
	xBoxFlag 							:BOOL;
	BoxBuffer							:BoxBufferHandling;
	ClearBoxBuffer_Rtrig				:R_TRIG;
	iTool_Num							:INT;
	fbSetToolTransform  				:L_MC4P_SetToolTransform;
	fbSetActiveTool						:L_MC4P_SetActiveTool;
	ToolRef								:L_MC4P_TOOL_REF;
    iSetToolStep						:INT;
	xSetToolDone						:BOOL;
	PickReadyCount						:INT;
	iWaitConditionJump					:INT:=6;//最近的抓取指令行
	//iNoJumpCount						:INT;
	//------------------------authorize ------------------//
	
	bValid_Lic_Type						: Lic_Type;
	bValid_Basic						: BOOL;
	bValid_MultiPick					: BOOL;
	bValid_LoadBalance					: BOOL;
	bValid_FASTlic						: BOOL;
	lrPickAuxC							: LREAL;
	lrNextProdPickAuxC  				: LREAL;
	//------------------------authorize ------------------//

	//Multipick
	fb_ProductCoordTransform			: L_RPP_ProductCoordTransform;
	iSelectSuckerNum					: INT;//选定的吸盘号
	i									: INT;
	wPickWithBeltStep_PCS_7				: WORD;
	wPickWithBeltStep_PCS_8				: WORD;
	wPickWithBeltStep_PCS_9				: WORD;
	                                	
	//Place 变址功能累加数                 	
	iAddPtNum							: INT;//变址累加数值
	//******************************************************************************                			
	fbPT1Filter_1									: L_USPP_PT1Filter;	
	lrDelayTime										: LREAL:=1.0;		
	lrInfeederActVelocity							: LREAL;	
	lrFactor										: LREAL:=0.2;
	lrTimeOfProdArrived								: LREAL;
	lrMinClutchTime									: LREAL:=0.12;		
	fb_BoxMoveEnable_TON							:TON;
	lrHeightCoefficient			: LREAL:=0.16;
	iPalletRow										:INT:=16;//托盘行数
	iPalletColumn									:INT:=16;//托盘列数
	iPick_Index										:INT; // 抓取索引
	iPick_Row										:INT; // 抓取行索引
	iPick_Column									:INT; // 抓取列索引
	iPlace_Index									:INT; // 放置索引
	iPlace_Row										:INT; // 放置行索引
	iPlace_Column									:INT; // 放置列索引
	iMotionLaw										:INT:=3;	
	ascPnPData_store								:ARRAY [1..256] OF scPnP_Data;//存储上位机发送数据信息
	iPnPData_index									:INT:=1;//用于检索ascPnPData_store中的数据
	scDataInformation_FromSiemens					:scDataMotion_FromSiemens;// Struct Interface from PLC
	scDataInformation_ToSiemens		    			:scDataMotion_ToSiemens;// Struct Interface to PLC 
 	iPickNr											:INT;//等待事件2中解析出来的抓取索引
	iPlaceNr										:INT;//等待事件2中解析出来的放置索引
	iUseDeltaDis									:INT:=1;//是否启用偏移量 7.5*rPalletPickDeltaX
	fb_DetectRunStart								:R_TRIG;// 检测开始启动上升沿
	eRobotState_to_UpPLC			:eSlaveToMaster_State;//将状态转换传递给上位机 2018.03.08
END_VAR

//将scDataInformation_FromSiemens、scDataInformation_ToSiemens结构体置于PLC的每个扫描周期内 
	IF scDataInformation_FromSiemens.scDataMotionFromPLC.wCtrl_2.wCtrl_scWord_to_bits1.xbit1=TRUE THEN
		 ;
	 END_IF
	 IF scDataInformation_ToSiemens.scDataMotionToPLC.wCtrl_16.wCtrl_scWord_to_bits1.xbit1=TRUE THEN
		 ;
	 END_IF
	
 //将scDataInformation_FromSiemens、scDataInformation_ToSiemens结构体置于PLC的每个扫描周期内
IF xEnable THEN				
	//7. 抓取模块报错
	IF L_RPP_PickPlace_0.ErrorID<>0 THEN
		ErrorID:=L_RPP_PickPlace_0.ErrorID;
	END_IF
	
	IF L_RPP_PickPlace_1.ErrorID<>0 THEN
		ErrorID:=L_RPP_PickPlace_1.ErrorID;
	END_IF
			
	IF ErrorID<>0 THEN
		xRunOrStopPrg:=FALSE;
		xRunPermission:=FALSE;
	END_IF	
			
	//开始或继续运动
	IF xRunOrStopPrg AND xChangeMotionType THEN		
		fb_TON_ResetPnP.IN:=TRUE;
		fb_TON_ResetPnP.PT:=T#50MS;
		xPnPReset:=TRUE;
	END_IF
	
	//PnP模块复位
	IF fb_TON_ResetPnP.Q THEN 
		xPnPReset:=FALSE;
		fb_TON_ResetPnP.IN:=FALSE;
		xRunPermission:=TRUE;
		MC_TrackConveyorBelt_U1.Abort:=FALSE;
	END_IF
		
	//开始启动上升沿 2018.3.5
	fb_DetectRunStart(CLK:=xRunOrStopPrg , Q=> );//开始启动上升沿 2018.3.5

	IF fb_DetectRunStart.Q THEN
		iCurrentPrgCmdNum:=iStartPrgCmdNum; //一旦启动开始，从指定行运行 2018.3.5
		iPnPData_index:=iBufferLine_HMI;//用示教器上的数值iBufferLine_HMI对iPnPDataIndex进行赋值操作,中途出错只能从Pick开始！
	END_IF
	//开始启动上升沿 2018.3.5
	
	//只有在当前运动行结束之后才可以停止运动
	IF (NOT	xRunOrStopPrg ) AND xChangeMotionType THEN
		xRunPermission:=FALSE;
		MC_TrackConveyorBelt_U1.Execute:=FALSE;
		MC_TrackConveyorBelt_U1.ClutchTimeAbort:=0.2;
		MC_TrackConveyorBelt_U1.Abort:=TRUE;
	END_IF 	
	
	A00_ProgramHandling();// 用户程序处理	
	
	IF xResetAutoRun   THEN
		xRunPermission:=FALSE;
	END_IF
	
END_IF


fb_TON_Dur1();		
IF fb_TON_Dur1.Q=TRUE THEN  //对外输出信号复位
	fb_TON_Dur1.IN:=FALSE;
	iOutputVal:=0;
END_IF

TOF_PrDel();
fb_TON_Delay();
TOF_BoxFull();
fb_TON_ResetPnP();			
fb_P2P(AxesGroup:=Delta_Robot);
fb_MoveLinear(AxesGroup:=Delta_Robot);
fb_MoveCircle(AxesGroup:=Delta_Robot);				
//自定义模块复位接口

MoveToWaitPoint0.Reset:=xPnPReset;	
L_RPP_PickPlace_0.Reset:=xPnPReset;
L_RPP_PickPlace_1.Reset:=xPnPReset;

L_RPP_PickPlace_0( AxesGroup:=Delta_Robot ); 
L_RPP_PickPlace_1( AxesGroup:=Delta_Robot );
MoveToWaitPoint0( AxesGroup:=Delta_Robot,Aux1:=AuxC );	

Robot_Stop( AxesGroup:=Delta_Robot);//轴组Stop
AuxC_Stop(Axis:=AuxC);//电机轴Stop			
fb_TON();

//PaP运动出错处理
IF  Delta_Robot.xError THEN	
	AuxC_Stop.Execute:=TRUE;
END_IF		

IF AuxC_Stop.Done THEN
	AuxC_Stop.Execute:=FALSE;
END_IF		

IF AuxC.xError THEN
	Robot_Stop.Execute:=TRUE;
END_IF

IF Robot_Stop.Done THEN
	Robot_Stop.Execute:=FALSE;
END_IF
//PaP运动出错处理

Run_RTrig(CLK:=xRunInter, Q=>);
Stop_RTrig(CLK:=xStopInter, Q=>);

IF 	Run_RTrig.Q THEN
	xRunOrStopPrg:=TRUE;
END_IF
IF 	Stop_RTrig.Q THEN
	xRunOrStopPrg:=FALSE;
END_IF			
			
Pick0_RTrig(CLK:=L_RPP_PickPlace_0.SWOut, Q=>);
Pick1_RTrig(CLK:=L_RPP_PickPlace_1.SWOut, Q=>);	

IF Pick0_RTrig.Q AND (iSuckDiscNr=1 OR iSuckDiscNr=0 ) THEN
	xSuckInter:=TRUE; xSuckInter2:=TRUE;
END_IF	

IF Pick0_RTrig.Q AND iSuckDiscNr=2 THEN //吸盘2 控制
	xSuckInter2:=TRUE;
END_IF	

IF Pick1_RTrig.Q THEN
	xBlowInter:=TRUE;
END_IF	

IF xBlowInter THEN
	xSuckInter:=FALSE; 
	xSuckInter2:=FALSE;
	fb_TON3.IN:=TRUE;
	fb_TON3.PT:=REAL_TO_TIME(rBlowGasTime);//是否是MS？
END_IF
	
IF fb_TON3.Q=TRUE THEN
	xBlowInter:=FALSE;
	fb_TON3.IN:=FALSE;
	//xSuckBlowLock:=TRUE;				
END_IF
xSuck:=xSuckInter;
xSuck2:=xSuckInter2; //吸盘2
xBlow:=xBlowInter;
fb_TON3();
		
		
IF NOT xEnable	 THEN
	//Step 回零
	iPickedPrdNr:=0;
	iCurrentPrgCmdNum:=1;
	xBlowInter:=FALSE;
	xSuckInter:=FALSE;
	xSuckInter2:=FALSE;
	//Step 回零
	iAutoStep:=0;
	wPickAloneStep:=0;		
	wPickWithBeltStep:=0;	
	wPickWithBeltStep_PCS_7:=0;
	wPickWithBeltStep_PCS_8:=0;
	wPickWithBeltStep_PCS_9:=0;			
	wPlaceAloneStep:=0;	
	wPlaceWithBeltStep:=0;
	wPlaceSafeStep:=0;
	//启动回零
	xRunOrStopPrg:=FALSE;
	//运动模块执行初始化
	fb_P2P.Execute:=FALSE;//P2P中途出错复位
	fb_MoveLinear.Execute:=FALSE;
	fb_MoveCircle.Execute:=FALSE;
	L_RPP_PickPlace_0.Execute:=FALSE; 
	L_RPP_PickPlace_1.Execute:=FALSE;
	MoveToWaitPoint0.Execute:=FALSE;
	fb_TON.IN:=FALSE;
	MC_TrackConveyorBelt_U1.Execute:=FALSE;
	MC_TrackConveyorBelt_U1.ClutchTimeAbort:=0.2;
	MC_TrackConveyorBelt_U1.Abort:=TRUE;
	MC_TrackConveyorBelt_U2.Execute:=FALSE;
	MC_TrackConveyorBelt_U2.ClutchTimeAbort:=0.2;
	MC_TrackConveyorBelt_U2.Abort:=TRUE;
	FOR i:=1 TO 10 BY 1 DO
		MC_TrackConveyorBelt_U[i].Execute:=FALSE;
		MC_TrackConveyorBelt_U[i].Abort:=TRUE;
		MC_TrackConveyorBelt_U[i].ClutchTimeAbort:=0.2;
	END_FOR
	//清空Jump中的跳转次数
	SysMemSet(pDest:=ADR(aiJumpCount) , udiValue:=0 , udiCount:=SIZEOF(aiJumpCount) );
	//执行逻辑初始化
	iCurrentPrgCmdNum:=1;
	iCommandType:=0;
	xChangeMotionType:=TRUE;
	// ErrorID复位
	// ErrorID:=0 ;
	xBoxFlag:=0;
	iJumpCount:=0;
	xSearchPlaceCmd:=FALSE;
	//xNew_Place:=FALSE;
	xWarning:=FALSE;
	AuxC_Stop.Execute:=FALSE;//Stop功能块复位
	Robot_Stop.Execute:=FALSE;//Stop功能块复位
	xBoxMoveEnable:=TRUE;
	
END_IF

IF xResetAutoRun THEN
	iPickedPrdNr:=0;
	iCurrentPrgCmdNum:=1;
	xBlowInter:=FALSE;
	xSuckInter:=FALSE;
	xSuckInter2:=FALSE;
	//Step 回零
	iAutoStep:=0;
	wPickAloneStep:=0;		
	wPickWithBeltStep:=0;	
	wPickWithBeltStep_PCS_7:=0;
	wPickWithBeltStep_PCS_8:=0;
	wPickWithBeltStep_PCS_9:=0;			
	wPlaceAloneStep:=0;	
	wPlaceWithBeltStep:=0;
	wPlaceSafeStep:=0;
	//启动回零
	xRunOrStopPrg:=FALSE;
	//运动模块执行初始化
	fb_P2P.Execute:=FALSE;//P2P中途出错复位
	fb_MoveLinear.Execute:=FALSE;
	fb_MoveCircle.Execute:=FALSE;
	L_RPP_PickPlace_0.Execute:=FALSE; 
	L_RPP_PickPlace_1.Execute:=FALSE;
	MoveToWaitPoint0.Execute:=FALSE;
	fb_TON.IN:=FALSE;
	MC_TrackConveyorBelt_U1.Execute:=FALSE;
	MC_TrackConveyorBelt_U1.ClutchTimeAbort:=0.2;
	MC_TrackConveyorBelt_U1.Abort:=TRUE;
	MC_TrackConveyorBelt_U2.Execute:=FALSE;
	MC_TrackConveyorBelt_U2.ClutchTimeAbort:=0.2;
	MC_TrackConveyorBelt_U2.Abort:=TRUE;
	FOR i:=1 TO 10 BY 1 DO
		MC_TrackConveyorBelt_U[i].Execute:=FALSE;
		MC_TrackConveyorBelt_U[i].Abort:=TRUE;
		MC_TrackConveyorBelt_U[i].ClutchTimeAbort:=0.2;
	END_FOR
	//清空Jump中的跳转次数
	SysMemSet(pDest:=ADR(aiJumpCount) , udiValue:=0 , udiCount:=SIZEOF(aiJumpCount) );
	//执行逻辑初始化
	iCurrentPrgCmdNum:=1;
	iCommandType:=0;
	xChangeMotionType:=TRUE;
	// ErrorID复位
	// ErrorID:=0 ;
	xBoxFlag:=0;
	iJumpCount:=0;
	xSearchPlaceCmd:=FALSE;
	//xNew_Place:=FALSE;
	xWarning:=FALSE;
	AuxC_Stop.Execute:=FALSE;//Stop功能块复位
	Robot_Stop.Execute:=FALSE;//Stop功能块复位
	xBoxMoveEnable:=TRUE;
END_IF 

   
//	2016.11.30	
fb_ProductCoordTransform(Axis:=AuxC);

//2017.03.30
//L_RPP_TimeOfProdArrivedEvaluation_0(AxisConveyorBelt:=Infeeder);	
fbPT1Filter_1(
	lrIn:=Infeeder.lrActVelocity, 
	lrDelayTime:=lrDelayTime, 
	lrOut=>lrInfeederActVelocity, 
	xError=> ,
	eErrorID=> ); 

A03_RobotSateTransition();//将状态转换传递给上位机 2018.03.08

ACTION A01_PickAlone:
//=============================================================================
//xCameraEnable:=FALSE;//相机使能禁用

CASE wPickAloneStep OF
	0://	
		IF xRunOrStopPrg THEN
			wPickAloneStep:=50;
		END_IF
		
	//**************************************************************************	
	50://去抓取位置	
		//判断抓取位置是否是码盘抓取	
		iPick_Row:=0;    //初始化
		iPick_Column:=0; //初始化		
		
		//若抓取点号为1，设置抓取坐标系为PCS5
		IF CustomerPrg.Table_Command_Pick[iCommandIndex].iPtNo=1 THEN
			L_RPP_PickPlace_0.CoordSystem:=L_MC4P_CoordSystem.PCS_5;
		ELSIF CustomerPrg.Table_Command_Pick[iCommandIndex].iPtNo=2 THEN
			L_RPP_PickPlace_0.CoordSystem:=L_MC4P_CoordSystem.PCS_6;	
		ELSE
			L_RPP_PickPlace_0.CoordSystem:=CustomerPrg.Table_Position[CustomerPrg.Table_Command_Pick[iCommandIndex].iPtNo].CS_Num;	//用户设置联系变量			
		END_IF	
		//若抓取点号为1，设置抓取坐标系为PCS5	
		
		IF xExternalMode=TRUE THEN
			iPick_Index:=iPickNr;
			//L_RPP_PickPlace_0.CoordSystem:=L_MC4P_CoordSystem.PCS_5;//若为外部模式，强制转换坐标系
		ELSE
			iPick_Index:=CustomerPrg.Table_Command_Pick[iCommandIndex].iPnP_Index;	//码盘索引号
		END_IF
		
		IF CustomerPrg.Table_Command_Pick[iCommandIndex].iPtNo=1 OR CustomerPrg.Table_Command_Pick[iCommandIndex].iPtNo=2 THEN //如果抓取点为1，则激活索引功能
			iPick_Row:=LREAL_TO_INT((iPick_Index-1)/iPalletRow); //PCS X方向
			iPick_Column:=(iPick_Index-1) MOD iPalletColumn;	 //PCS Y方向
			iUseDeltaDis:=1;
		ELSE
			iUseDeltaDis:=0;
		END_IF				 
		//判断抓取位置是否是码盘抓取					
		L_RPP_PickPlace_0.TargetPosition[1]:= CustomerPrg.Table_Position[CustomerPrg.Table_Command_Pick[iCommandIndex].iPtNo].X+iPick_Row*rPalletPickDeltaX-7.5*rPalletPickDeltaX*iUseDeltaDis;		
		L_RPP_PickPlace_0.TargetPosition[2]:= CustomerPrg.Table_Position[CustomerPrg.Table_Command_Pick[iCommandIndex].iPtNo].Y+iPick_Column*rPalletPickDeltaY-7.5*rPalletPickDeltaY*iUseDeltaDis;	
		L_RPP_PickPlace_0.TargetPosition[3]:= CustomerPrg.Table_Position[CustomerPrg.Table_Command_Pick[iCommandIndex].iPtNo].Z+rSuckerDropHeight;//气阀下降高度		
		L_RPP_PickPlace_0.TargetPosition[7]:= CustomerPrg.Table_Position[CustomerPrg.Table_Command_Pick[iCommandIndex].iPtNo].C;		
		L_RPP_PickPlace_0.StartHeight:=CustomerPrg.Table_Command_Pick[iCommandIndex].rH1; //10
		L_RPP_PickPlace_0.TargetHeight:=CustomerPrg.Table_Command_Pick[iCommandIndex].rH2;
		L_RPP_PickPlace_0.Duration:=CustomerPrg.Table_Command_Pick[iCommandIndex].rMovTime;  //Unit:s	0.5			
		L_RPP_PickPlace_0.HeightCoefficient:=lrHeightCoefficient;
		L_RPP_PickPlace_0.SwitchTime:=rSuckOpenTime/1000.0; //0.1		
		L_RPP_PickPlace_0.iReParaLaw:=iMotionLaw;	
		L_RPP_PickPlace_0.xDuraCondition:=(iSelfadaptPickSwitch=1);
		IF iSelfadaptPickSwitch=1 THEN
			L_RPP_PickPlace_0.DurationRange[1]:=rPnPDurationNegativeLimit;
			L_RPP_PickPlace_0.DurationRange[2]:=rPnPDurationPositiveLimit;
		END_IF		
		L_RPP_PickPlace_0.Execute:= TRUE;
		wPickAloneStep:=60;			
	60://
		IF L_RPP_PickPlace_0.Busy THEN
			L_RPP_PickPlace_0.Execute:= FALSE;
			wPickAloneStep:=80;	
		END_IF	
	
	80://		
		IF L_RPP_PickPlace_0.Done THEN	
			wPickAloneStep:=0;
			xDoNextCmd:=TRUE;
		END_IF
END_CASE
END_ACTION

ACTION A02_PlaceAlone:

CASE wPlaceAloneStep OF				
	0://返回初始位置	
		//判断抓取位置是否是码盘抓取	
		iPlace_Row:=0;    //初始化
		iPlace_Column:=0; //初始化
		
		//若抓取点号为1，设置抓取坐标系为PCS6
		IF CustomerPrg.Table_Command_Place[iCommandIndex].iPtNo=1 THEN
			L_RPP_PickPlace_1.CoordSystem:=L_MC4P_CoordSystem.PCS_5;			
		ELSIF CustomerPrg.Table_Command_Place[iCommandIndex].iPtNo=2 THEN
			L_RPP_PickPlace_1.CoordSystem:=L_MC4P_CoordSystem.PCS_6;			
		ELSE
			L_RPP_PickPlace_1.CoordSystem:=CustomerPrg.Table_Position[CustomerPrg.Table_Command_Place[iCommandIndex].iPtNo].CS_Num;	//用户设置联系变量			
		END_IF		
		//若抓取点号为1，设置抓取坐标系为PCS6
		
		IF xExternalMode=TRUE THEN
			iPlace_Index:=iPlaceNr;
			//L_RPP_PickPlace_1.CoordSystem:=L_MC4P_CoordSystem.PCS_6;//若为外部模式，强制转换坐标系
		ELSE
			iPlace_Index:=CustomerPrg.Table_Command_Place[iCommandIndex].iPnP_Index;	//码盘索引号
		END_IF		
		
	
		IF CustomerPrg.Table_Command_Place[iCommandIndex].iPtNo=1 OR CustomerPrg.Table_Command_Place[iCommandIndex].iPtNo=2 THEN //如果抓取点为1，则激活索引功能
			iPlace_Row:=LREAL_TO_INT((iPlace_Index-1)/iPalletRow); //PCS X方向
			iPlace_Column:=(iPlace_Index-1) MOD iPalletColumn;	   //PCS Y方向	
			iUseDeltaDis:=1;
		ELSE
			iUseDeltaDis:=0;	
		END_IF				 
		//判断抓取位置是否是码盘抓取
		
				
	
		//放置目标计算	
		L_RPP_PickPlace_1.TargetPosition[1]:=CustomerPrg.Table_Position[CustomerPrg.Table_Command_Place[iCommandIndex].iPtNo].X+iPlace_Row*rPalletPickDeltaX-7.5*rPalletPickDeltaX*iUseDeltaDis;
		L_RPP_PickPlace_1.TargetPosition[2]:=CustomerPrg.Table_Position[CustomerPrg.Table_Command_Place[iCommandIndex].iPtNo].Y+iPlace_Column*rPalletPickDeltaY-7.5*rPalletPickDeltaY*iUseDeltaDis;
		L_RPP_PickPlace_1.TargetPosition[3]:=CustomerPrg.Table_Position[CustomerPrg.Table_Command_Place[iCommandIndex].iPtNo].Z;
		L_RPP_PickPlace_1.TargetPosition[7]:=CustomerPrg.Table_Position[CustomerPrg.Table_Command_Place[iCommandIndex].iPtNo].C;
		L_RPP_PickPlace_1.StartHeight:=CustomerPrg.Table_Command_Place[iCommandIndex].rH1; //h1
		L_RPP_PickPlace_1.TargetHeight:=CustomerPrg.Table_Command_Place[iCommandIndex].rH2;	//h2
		//L_RPP_PickPlace_1.AccDecTimeRatio:=CustomerPrg.Table_Command_Place[iCommandIndex].rAcc2Dec; //加速减速比
		L_RPP_PickPlace_1.Duration:=CustomerPrg.Table_Command_Place[iCommandIndex].rMovTime;  //Unit:s	MoveCycleTime
		L_RPP_PickPlace_1.SwitchTime:=rBlowOpenTime/1000.0;//0.1
		L_RPP_PickPlace_1.HeightCoefficient:=lrHeightCoefficient;
		
		L_RPP_PickPlace_1.iReParaLaw:=iMotionLaw; // 1 加减速为1:1  //2 加减速为4.5:5.5  //3  加减速为4:6
		L_RPP_PickPlace_1.xDuraCondition:=(iSelfadaptPickSwitch=1);
		IF iSelfadaptPickSwitch=1 THEN
			L_RPP_PickPlace_1.DurationRange[1]:=rPnPDurationNegativeLimit;
			L_RPP_PickPlace_1.DurationRange[2]:=rPnPDurationPositiveLimit;
		END_IF
		
			
		L_RPP_PickPlace_1.Execute:= TRUE;		

		IF ErrorID=0 THEN
			wPlaceAloneStep:=10;
		END_IF

	10://	
		IF L_RPP_PickPlace_1.Busy THEN
			L_RPP_PickPlace_1.Execute:= FALSE;	
			wPlaceAloneStep:=20;	
		END_IF	
		
	20://
		IF L_RPP_PickPlace_1.Done THEN			
			wPlaceAloneStep:=0;
			xDoNextCmd:=TRUE;
			BoxBuffer.xPlaceRunning:=FALSE;//如果完成装箱，告知BoxBuffer，Place结束！
		END_IF
END_CASE
END_ACTION

ACTION A00_ProgramHandling:
IF xRunPermission  AND ErrorID=0 THEN //如果出现ErrorID则系统会停止运行	
	
	IF xBoxMoveEnable=TRUE THEN
		fb_BoxMoveEnable_TON.IN:=TRUE;
	ELSE
		fb_BoxMoveEnable_TON.IN:=FALSE;
	END_IF
	
	IF fb_BoxMoveEnable_TON.Q THEN
		xBoxMoveEnable:=FALSE;
	END_IF
	
	iCommandType:=CustomerPrg.Table_Clause[iCurrentPrgCmdNum].CommandType;
	iCommandIndex:=CustomerPrg.Table_Clause[iCurrentPrgCmdNum].CommandIndex;
	
	IF 	xChangeMotionType=TRUE THEN //当前程序执行完毕可以将类型赋给下一运动类型
		iAutoStep:=iCommandType;
		xChangeMotionType:=FALSE;
	END_IF
															
	CASE iAutoStep OF
		0:
			xDoNextCmd:=TRUE;
		1:									//P2P
			IF CustomerPrg.Table_Command_P2P[iCommandIndex].iPtNo<>0 THEN
				fb_P2P.CoordSystem:=L_MC4P_CoordSystem.MCS;  
				fb_P2P.Position[1]:=CustomerPrg.Table_Position[CustomerPrg.Table_Command_P2P[iCommandIndex].iPtNo].X;
				fb_P2P.Position[2]:=CustomerPrg.Table_Position[CustomerPrg.Table_Command_P2P[iCommandIndex].iPtNo].Y;
				fb_P2P.Position[3]:=CustomerPrg.Table_Position[CustomerPrg.Table_Command_P2P[iCommandIndex].iPtNo].Z;
				fb_P2P.Position[7]:=CustomerPrg.Table_Position[CustomerPrg.Table_Command_P2P[iCommandIndex].iPtNo].C;					
				fb_P2P.Execute:=TRUE;						
				iAutoStep:=11;	
			ELSE
				ErrorID:=30201;
			END_IF
										
		2:									//MoveLinear
			IF CustomerPrg.Table_Command_MoveLinear[iCommandIndex].iPtNo<>0 AND CustomerPrg.Table_Command_MoveLinear[iCommandIndex].rVel<>0 THEN
				fb_MoveLinear.CoordSystem:=L_MC4P_CoordSystem.MCS;
				fb_MoveLinear.Position[1]:=CustomerPrg.Table_Position[CustomerPrg.Table_Command_MoveLinear[iCommandIndex].iPtNo].X;
				fb_MoveLinear.Position[2]:=CustomerPrg.Table_Position[CustomerPrg.Table_Command_MoveLinear[iCommandIndex].iPtNo].Y;
				fb_MoveLinear.Position[3]:=CustomerPrg.Table_Position[CustomerPrg.Table_Command_MoveLinear[iCommandIndex].iPtNo].Z;
				fb_MoveLinear.Position[7]:=CustomerPrg.Table_Position[CustomerPrg.Table_Command_MoveLinear[iCommandIndex].iPtNo].C;									
				fb_MoveLinear.Velocity:=CustomerPrg.Table_Command_MoveLinear[iCommandIndex].rVel; //速度单位不一致需修改
				fb_MoveLinear.Acceleration:=100;
				fb_MoveLinear.Deceleration:=100;
				fb_MoveLinear.Jerk:=10000;
				//fb_MoveLinear.aeAuxMode[1]:=L_MC4P_AuxMode.Continuous;//辅助与主轴连续运动     连续运动movelinear执行卡住，功能块还需测试
				fb_MoveLinear.Execute:=TRUE;
				iAutoStep:=12;
			ELSE
				ErrorID:=30202;
			END_IF
			
		3:									//MoveCircle
			IF CustomerPrg.Table_Command_MoveCircle[iCommandIndex].iPt1No<>0 AND  CustomerPrg.Table_Command_MoveCircle[iCommandIndex].iPt2No<>0 
						AND  CustomerPrg.Table_Command_MoveCircle[iCommandIndex].rVel<>0 THEN
				fb_MoveCircle.CoordSystem:=L_MC4P_CoordSystem.MCS;
				fb_MoveCircle.AuxPoint[1]:= CustomerPrg.Table_Position[CustomerPrg.Table_Command_MoveCircle[iCommandIndex].iPt1No].X;
				fb_MoveCircle.AuxPoint[2]:= CustomerPrg.Table_Position[CustomerPrg.Table_Command_MoveCircle[iCommandIndex].iPt1No].Y;                  								
				fb_MoveCircle.AuxPoint[3]:= CustomerPrg.Table_Position[CustomerPrg.Table_Command_MoveCircle[iCommandIndex].iPt1No].Z;                  								
				fb_MoveCircle.AuxPoint[7]:= CustomerPrg.Table_Position[CustomerPrg.Table_Command_MoveCircle[iCommandIndex].iPt1No].C;                  								
				fb_MoveCircle.EndPoint[1]:= CustomerPrg.Table_Position[CustomerPrg.Table_Command_MoveCircle[iCommandIndex].iPt2No].X;                  								
				fb_MoveCircle.EndPoint[2]:= CustomerPrg.Table_Position[CustomerPrg.Table_Command_MoveCircle[iCommandIndex].iPt2No].Y;                  								
				fb_MoveCircle.EndPoint[3]:= CustomerPrg.Table_Position[CustomerPrg.Table_Command_MoveCircle[iCommandIndex].iPt2No].Z;                  								
				fb_MoveCircle.EndPoint[7]:= CustomerPrg.Table_Position[CustomerPrg.Table_Command_MoveCircle[iCommandIndex].iPt2No].C;
				fb_MoveCircle.CircMode:=L_MC4P_CircMode.BORDER;                 								
				fb_MoveCircle.PathChoice:=MC_CIRC_PATHCHOICE.CLOCKWISE;
				fb_MoveCircle.Velocity:=CustomerPrg.Table_Command_MoveCircle[iCommandIndex].rVel;
				fb_MoveCircle.Acceleration:=100;
				fb_MoveCircle.Deceleration:=100;
				fb_MoveCircle.Jerk:=1000;
				//fb_MoveCircle.aeAuxMode[1]:=L_MC4P_AuxMode.Continuous;//辅助与主轴连续运动
				fb_MoveCircle.Execute:=TRUE;
				iAutoStep:=13;			
			ELSE	
				ErrorID:=30203;
			END_IF
																
			
		4:	//Pick
			//eRobotState_to_UpPLC:=eSlaveToMaster_State.Running;//机器人进入运行状态 03.08
			
			IF CustomerPrg.Table_Command_Pick[iCommandIndex].iPtNo<>0 AND CustomerPrg.Table_Command_Pick[iCommandIndex].rMovTime<>0 THEN
	
				A01_PickAlone();		
			ELSE
				ErrorID:=30204;  
			END_IF
								
		5:	//Place
			//eRobotState_to_UpPLC:=eSlaveToMaster_State.Running;//机器人进入运行状态 03.08
			
			IF CustomerPrg.Table_Command_Place[iCommandIndex].iPtNo<>0 AND CustomerPrg.Table_Command_Place[iCommandIndex].rMovTime<>0 THEN
	
				A02_PlaceAlone();																						
			ELSE 
				ErrorID:=30205;  
			END_IF
											
		6:		//MoveWaitPoint
			IF CustomerPrg.Table_Command_MoveWaitPoint[iCommandIndex].rMovTime<>0 AND CustomerPrg.Table_Command_MoveWaitPoint[iCommandIndex].rH<>0 THEN
				
				IF CustomerPrg.Table_Clause[iCurrentPrgCmdNum+1].CommandType=L_RPP_CommandType.Pick THEN //如果下一条指令是抓取，则变换角度
					
					//lrNextProdPickAuxC:=lrNextProdAuxC;												
					IF ABS(lrNextProdAuxC)<=90 THEN
						lrNextProdPickAuxC:=lrNextProdAuxC;
					ELSIF lrNextProdAuxC<-90 THEN
						lrNextProdPickAuxC:=180+lrNextProdAuxC;		
					ELSIF lrNextProdAuxC>90 THEN
						lrNextProdPickAuxC:=lrNextProdAuxC-180;		
					END_IF
				ELSE
					lrNextProdPickAuxC:=1;	
				END_IF
	
	
				MoveToWaitPoint0.Duration:=CustomerPrg.Table_Command_MoveWaitPoint[iCommandIndex].rMovTime;
				MoveToWaitPoint0.TargetPosition[3]:= CustomerPrg.Table_Command_MoveWaitPoint[iCommandIndex].rH;
				MoveToWaitPoint0.TargetPosition[7]:=lrNextProdPickAuxC;
				
				MoveToWaitPoint0.Execute:=TRUE;		
				MoveToWaitPoint0.CoordSystem:=L_MC4P_CoordSystem.MCS;              //2016.10.17修订
				//MoveToWaitPoint0.ConveyorBeltVelocity:=Outfeeder.lrActVelocity;    //2016.10.17修订         
				//MoveToWaitPoint0.DeclutchTime:=rOutfeedClutchPra*0.5;				 //2016.10.17修订
				iAutoStep:=16;												
			ELSE	
				ErrorID:=30206;  
			END_IF
	
		7:	
			//eRobotState_to_UpPLC:=eSlaveToMaster_State.Waiting;//机器人进入待机状态 03.08
			
			//1.WaitEvent接收外部信号的处理机制
			IF CustomerPrg.Table_Command_WaitEvent[iCommandIndex].iExternalEvent=5 OR 
				CustomerPrg.Table_Command_WaitEvent[iCommandIndex].iExternalEvent=6
				OR CustomerPrg.Table_Command_WaitEvent[iCommandIndex].iExternalEvent=7 THEN			
				iExtWaitEventNum:=	CustomerPrg.Table_Command_WaitEvent[iCommandIndex].iExternalEvent;	//WaitEvent 定义内部/外部事件成立？	
			END_IF
			//2.WaitEvent接收内部信号的处理机制
			iInterWaitEventNum:=CustomerPrg.Table_Command_WaitEvent[iCommandIndex].iInternalEvent;//内部事件编号
			iInterEventJumpNo:=CustomerPrg.Table_Command_WaitEvent[iCommandIndex].iInternalJump_No;//内部跳转行号
								
			//2.1 内部事件1--如果接收到上位机传递信息状态位，将数据全部存入	ascPnPData_store[1~256]	中  2018.3.1
			IF iInterWaitEventNum=1 THEN
				j:=1;													   											
				IF scDataInformation_FromSiemens.scDataMotionFromPLC.wCtrl_2.wCtrl_scWord_to_bits1.xbit1=TRUE THEN //上位机传递的状态信息
					
					iPnPData_index:=1;	//对iPnPData_index进行复位					
					SysMemSet(pDest:=ADR(ascPnPData_store),udiValue:=0,udiCount:=SIZEOF(ascPnPData_store));//清空ascPnPData_store数据信息
	
					FOR i:=1 TO 256 DO
						IF scDataInformation_FromSiemens.scDataMotionFromPLC.aPalletInformation[i]<>0 THEN
							ascPnPData_store[j].xStatus:=TRUE;
							ascPnPData_store[j].iPickPosition:=i;
							ascPnPData_store[j].iPlacePosition:=WORD_TO_INT(scDataInformation_FromSiemens.scDataMotionFromPLC.aPalletInformation[i]);
							j:=j+1;
						END_IF
					END_FOR			
					
					//scDataInformation_ToSiemens.scDataMotionToPLC.dwStatW1.xbit1:=TRUE;//机器人传递的读取状态信息					
					xDoNextCmd:=TRUE;					
				END_IF													
			END_IF
			
			//2.2 内部事件2--调用存于ascPnPData_store中的抓取放置数据，若数据执行完毕，这直接跳转到指定行
			IF iInterWaitEventNum=2 THEN	
				
				IF ascPnPData_store[iPnPData_index].xStatus=TRUE THEN
					
					iBufferLine_HMI:=iPnPData_index; //将正在调用的索引显示到示教器上
					
					iPickNr:=ascPnPData_store[iPnPData_index].iPickPosition;
					iPickRow_HMI:=LREAL_TO_INT((iPnPData_index-1)/iPalletRow); //Pick PCS X方向
					iPickCol_HMI:=(iPnPData_index-1) MOD iPalletColumn;	      //Pick PCS Y方向
					
					iPlaceNr:=ascPnPData_store[iPnPData_index].iPlacePosition;
					iPlaceRow_HMI:=LREAL_TO_INT((iPnPData_index-1)/iPalletRow); //Place PCS X方向
					iPlaceCol_HMI:=(iPnPData_index-1) MOD iPalletColumn;	 //Place PCS Y方向	
					
					iPnPData_index:=iPnPData_index+1;//缓存索引加1，为下一个要检索的数值。
					
				ELSE
					iCurrentPrgCmdNum:=iInterEventJumpNo-1; //跳转到指定程序行
					iPnPData_index:=1;	//对iPnPData_index进行复位
					eRobotState_to_UpPLC:=eSlaveToMaster_State.MotionCompleted; //MotionCompleted-机器人进入完成状态 03.08 
					//scDataInformation_ToSiemens.scDataMotionToPLC.wCtrl_16.wCtrl_scWord_to_bits1.xbit5:=TRUE;//机器人传递的动作完成信息
					SysMemSet(pDest:=ADR(ascPnPData_store),udiValue:=0,udiCount:=SIZEOF(ascPnPData_store));//清空ascPnPData_store数据信息			
				END_IF	
				
				xDoNextCmd:=TRUE; 
				
			END_IF   
			
	
		8:									//WaitTime
			fb_TON.IN:= TRUE;
			t_waitime:= REAL_TO_TIME(CustomerPrg.Table_Command_WaitTime[iCommandIndex].rTime)*1000; //如果Time基本单位是ms的话？
			fb_TON.PT:= t_waitime; 
			iAutoStep:= 18;              								
		9:									//Jump
			IF CustomerPrg.Table_Command_Jump[iCommandIndex].iPrgLine<>0 THEN
				iPreJumpPrgNum:=iCurrentPrgCmdNum;//跳转前的程序行						
				iJumpTimes:=CustomerPrg.Table_Command_Jump[iCommandIndex].iCount;
				iJumpNum:=CustomerPrg.Table_Command_Jump[iCommandIndex].iPrgLine;
				iJumpOutInEvent:=CustomerPrg.Table_Command_Jump[iCommandIndex].iJumpOutInEvent;
				
				IF iJumpTimes<>0 THEN //iJumpTimes=0代表无限循环		
					aiJumpCount[iPreJumpPrgNum]:=aiJumpCount[iPreJumpPrgNum]+1;
					IF aiJumpCount[iPreJumpPrgNum]>=iJumpTimes THEN
						xDoNextCmd:=TRUE;
						aiJumpCount[iPreJumpPrgNum]:=0;//跳转计数复位
					ELSE
						iCurrentPrgCmdNum:=iJumpNum-1; //跳出后程序行自动加1，所以在此跳转行减1
						xDoNextCmd:=TRUE; 
					END_IF				
				ELSE
					iCurrentPrgCmdNum:=iJumpNum-1; //跳出后程序行自动加1，所以在此跳转行减1
					xDoNextCmd:=TRUE; 							
				END_IF
	
				//定义内部跳出条件，用于多抓一放
				IF iJumpOutInEvent=1 THEN
					IF xJumpEndCondition THEN	// 内部条件需要赋值！！							
						iCurrentPrgCmdNum:=iPreJumpPrgNum;//跳转前的程序行
						xDoNextCmd:=TRUE;
						xJumpEndCondition:=FALSE;
					END_IF
				END_IF
									
			ELSE
				ErrorID:=30209; 
			END_IF
			
		10:						//Output 实现功能 
			iOutputVal:=CustomerPrg.Table_Command_Output[iCommandIndex].xOutputVal;//输出外部信号Output
			iOutputDuration:=CustomerPrg.Table_Command_Output[iCommandIndex].iOutputDuration;
			iInputSignalNo:=CustomerPrg.Table_Command_Output[iCommandIndex].iInputSignalNo;//装箱结束判断
			xInputSetValue:=CustomerPrg.Table_Command_Output[iCommandIndex].xSetValue;
			
			IF iInputSignalNo=1 AND xInputSetValue=TRUE THEN
				xBoxFlag:=1; //判断是否是装箱
				//BoxBuffer.xPlaceBanExp:=FALSE;//启用装箱异常检测功能	
			END_IF
			IF iInputSignalNo=1 AND xInputSetValue=FALSE THEN
				xBoxFlag:=0; //判断是否是装箱
			END_IF
			
			IF iInputSignalNo=2 AND xInputSetValue=TRUE  THEN //对内输入信号决定是否删除箱体列表数据，内部为上升沿触发
				IF BoxBuffer.xPassedMaxLine=TRUE THEN//如果在删除箱体之前，箱体已经越界，则取消删除箱体
					BoxBuffer.xResetExcpt:=TRUE;//复位越界警告
				ELSE
					TOF_PrDel.IN:=TRUE;
					TOF_PrDel.PT:=T#10MS;	
					TOF_BoxFull.IN:=TRUE;
					TOF_BoxFull.PT:=T#1S;
				END_IF										
			END_IF
			
			IF iInputSignalNo=3 AND xInputSetValue=TRUE  THEN  //主机端启动出料带信号
				xMasterOutfeederStart:=TRUE;
			END_IF
			
			IF iInputSignalNo=4 AND xInputSetValue=TRUE  THEN //从机端启动出料带信号
				xSlaveOutfeederStart:=TRUE;
			END_IF
			
			IF iInputSignalNo=5 AND xInputSetValue=TRUE  THEN //清空装箱产品计数信号
				iPickedPrdNr:=0;	
			END_IF
			
			IF iOutputVal <>0 THEN
				fb_TON_Dur1.IN:=TRUE;
				fb_TON_Dur1.PT:=INT_TO_TIME(iOutputDuration);
			END_IF
			xDoNextCmd:=TRUE; 
		11:
			IF fb_P2P.Done=TRUE THEN
				fb_P2P.Execute:=FALSE;
				xDoNextCmd:=TRUE;
			END_IF
		12:
			IF fb_MoveLinear.Done=TRUE THEN
				fb_MoveLinear.Execute:=FALSE;
				xDoNextCmd:=TRUE;
			END_IF
		13:
			IF fb_MoveCircle.Done=TRUE THEN
				fb_MoveCircle.Execute:=FALSE;
				xDoNextCmd:=TRUE;
			END_IF	
		14:
	
		15:				
			
		16:	IF MoveToWaitPoint0.Done THEN
				MoveToWaitPoint0.Execute:=FALSE;
				xDoNextCmd:=TRUE;
			END_IF
	
		18:
			IF fb_TON.Q=TRUE THEN
				fb_TON.IN:=FALSE;
				xDoNextCmd:=TRUE;
			END_IF					
		25:					
	END_CASE
	
	IF xDoNextCmd AND iCurrentPrgCmdNum<=50 THEN //执行下一行
		iCurrentPrgCmdNum:=iCurrentPrgCmdNum+1;
		xDoNextCmd:=FALSE; 
		xChangeMotionType:=TRUE;
	END_IF	
	
	IF iCurrentPrgCmdNum>50 THEN //自动运行-执行完毕
		iCurrentPrgCmdNum:=1;
		xDoNextCmd:=FALSE;
		xChangeMotionType:=TRUE;
		//xAutoRun:=FALSE;
		xRunOrStopPrg:=FALSE;
	END_IF		
END_IF
END_ACTION

ACTION A03_RobotSateTransition:

IF xRunOrStopPrg=FALSE AND eRobotState_to_UpPLC<>eSlaveToMaster_State.Error THEN
	eRobotState_to_UpPLC:=eSlaveToMaster_State.Manual; //Manual-机器人进入手动状态 03.08
END_IF

IF iAutoStep=7 THEN
	eRobotState_to_UpPLC:=eSlaveToMaster_State.Waiting;//Waiting-机器人进入待机状态 03.08
END_IF

IF iAutoStep=4 OR iAutoStep=5 THEN
	eRobotState_to_UpPLC:=eSlaveToMaster_State.Running;//Running-机器人进入运行状态 03.08
END_IF

IF xSystemError OR xSystemWarning THEN
	eRobotState_to_UpPLC:=eSlaveToMaster_State.Error; //Error-机器人进入错误状态 03.08 
END_IF

//	wCtrl_scWord_to_bits1.xbit1 待机
//	wCtrl_scWord_to_bits1.xbit2 运行
//	wCtrl_scWord_to_bits1.xbit3 故障
//	wCtrl_scWord_to_bits1.xbit4 手动
//	wCtrl_scWord_to_bits1.xbit5 动作完成

IF xPnPReset=TRUE THEN //Reset
	scDataInformation_ToSiemens.scDataMotionToPLC.wCtrl_16.wCtrl_scWord_to_bits1.xbit1:=FALSE;
	scDataInformation_ToSiemens.scDataMotionToPLC.wCtrl_16.wCtrl_scWord_to_bits1.xbit2:=FALSE;
	scDataInformation_ToSiemens.scDataMotionToPLC.wCtrl_16.wCtrl_scWord_to_bits1.xbit3:=FALSE;
	scDataInformation_ToSiemens.scDataMotionToPLC.wCtrl_16.wCtrl_scWord_to_bits1.xbit4:=TRUE; 
END_IF

IF eRobotState_to_UpPLC=eSlaveToMaster_State.Manual THEN //Manual
	scDataInformation_ToSiemens.scDataMotionToPLC.wCtrl_16.wCtrl_scWord_to_bits1.xbit1:=FALSE;
	scDataInformation_ToSiemens.scDataMotionToPLC.wCtrl_16.wCtrl_scWord_to_bits1.xbit2:=FALSE;
	scDataInformation_ToSiemens.scDataMotionToPLC.wCtrl_16.wCtrl_scWord_to_bits1.xbit4:=TRUE; 
END_IF

IF eRobotState_to_UpPLC=eSlaveToMaster_State.Waiting THEN //Waiting
	scDataInformation_ToSiemens.scDataMotionToPLC.wCtrl_16.wCtrl_scWord_to_bits1.xbit1:=TRUE;
	scDataInformation_ToSiemens.scDataMotionToPLC.wCtrl_16.wCtrl_scWord_to_bits1.xbit2:=FALSE;
	scDataInformation_ToSiemens.scDataMotionToPLC.wCtrl_16.wCtrl_scWord_to_bits1.xbit4:=FALSE; 
END_IF

IF eRobotState_to_UpPLC=eSlaveToMaster_State.Running THEN //Running
	scDataInformation_ToSiemens.scDataMotionToPLC.wCtrl_16.wCtrl_scWord_to_bits1.xbit1:=FALSE;
	scDataInformation_ToSiemens.scDataMotionToPLC.wCtrl_16.wCtrl_scWord_to_bits1.xbit2:=TRUE;
	scDataInformation_ToSiemens.scDataMotionToPLC.wCtrl_16.wCtrl_scWord_to_bits1.xbit4:=FALSE; 
END_IF

IF eRobotState_to_UpPLC=eSlaveToMaster_State.MotionCompleted THEN //MotionCompleted 完成信号要有一定长度，上位机要截取上升沿
	scDataInformation_ToSiemens.scDataMotionToPLC.wCtrl_16.wCtrl_scWord_to_bits1.xbit5:=TRUE; 
END_IF

IF eRobotState_to_UpPLC=eSlaveToMaster_State.Error THEN //Error
	scDataInformation_ToSiemens.scDataMotionToPLC.wCtrl_16.wCtrl_scWord_to_bits1.xbit3:=TRUE;
END_IF
END_ACTION

END_PROGRAM

// Controller_3200C/Application/FunctionBlock/FourPts_Calibration
FUNCTION_BLOCK FourPts_Calibration

VAR_INPUT
	rReadfeedPos1_X		:REAL;
	rReadfeedPos1_Y 	:REAL;
	rReadfeedPos1_Z		:REAL;
	rReadfeedPos2_X		:REAL;
	rReadfeedPos2_Y		:REAL;
	rReadfeedPos3_X		:REAL;
	rReadfeedPos3_Y		:REAL;
	rReadfeedPos4_X		:REAL;
	rReadfeedPos4_Y		:REAL;
	n					:INT:=15;
END_VAR

VAR_OUTPUT
	rRotation_C			:REAL;
	Output_X0			:REAL;//PCS 下的X0坐标
	Output_Y0			:REAL;//PCS 下的Y0坐标
	Output_X1			:REAL;//PCS 下的X1坐标
	Output_Y1			:REAL;//PCS 下的Y1坐标
	Output_X2			:REAL;//PCS 下的X2坐标
	Output_Y2			:REAL;//PCS 下的Y2坐标
	Output_X3			:REAL;//PCS 下的X3坐标
	Output_Y3			:REAL;//PCS 下的Y3坐标
	dx					:REAL;//x方向间距
	dy					:REAL;//y方向间距
END_VAR

VAR
	rAngle_PI			:REAL;
	rAngle				:REAL;
	rAngle_a			:LREAL;
	rAngle_PI_a			:LREAL;
	rAngle_b			:LREAL;
	rAngle_PI_b			:LREAL;
	Tx,x0,x1,x2,x3		:REAL;
	Ty,y0,y1,y2,y3		:REAL;
	Tz					:REAL;
	C					:REAL;
END_VAR

IF (rReadfeedPos2_Y-rReadfeedPos1_Y)>=0 THEN
	rAngle:=360/(2*math.PI)*ACOS((rReadfeedPos2_X-rReadfeedPos1_X)/SQRT(EXPT((rReadfeedPos2_X-rReadfeedPos1_X),2)+EXPT((rReadfeedPos2_Y-rReadfeedPos1_Y),2)));
	rAngle_PI:=ACOS((rReadfeedPos2_X-rReadfeedPos1_X)/SQRT(EXPT((rReadfeedPos2_X-rReadfeedPos1_X),2)+EXPT((rReadfeedPos2_Y-rReadfeedPos1_Y),2)));
ELSE
	rAngle:=360-360/(2*math.PI)*ACOS((rReadfeedPos2_X-rReadfeedPos1_X)/SQRT(EXPT((rReadfeedPos2_X-rReadfeedPos1_X),2)+EXPT((rReadfeedPos2_Y-rReadfeedPos1_Y),2)));
	rAngle_PI:=2*math.PI-ACOS((rReadfeedPos2_X-rReadfeedPos1_X)/SQRT(EXPT((rReadfeedPos2_X-rReadfeedPos1_X),2)+EXPT((rReadfeedPos2_Y-rReadfeedPos1_Y),2)));;	
END_IF

IF (rReadfeedPos3_Y-rReadfeedPos1_Y)>=0 THEN
	rAngle_a:=360/(2*math.PI)*ACOS((rReadfeedPos3_X-rReadfeedPos1_X)/SQRT(EXPT((rReadfeedPos3_X-rReadfeedPos1_X),2)+EXPT((rReadfeedPos3_Y-rReadfeedPos1_Y),2)));
	rAngle_PI_a:=ACOS((rReadfeedPos3_X-rReadfeedPos1_X)/SQRT(EXPT((rReadfeedPos3_X-rReadfeedPos1_X),2)+EXPT((rReadfeedPos3_Y-rReadfeedPos1_Y),2)));
ELSE
	rAngle_a:=360-360/(2*math.PI)*ACOS((rReadfeedPos3_X-rReadfeedPos1_X)/SQRT(EXPT((rReadfeedPos3_X-rReadfeedPos1_X),2)+EXPT((rReadfeedPos3_Y-rReadfeedPos1_Y),2)));
	rAngle_PI_a:=2*math.PI-ACOS((rReadfeedPos3_X-rReadfeedPos1_X)/SQRT(EXPT((rReadfeedPos3_X-rReadfeedPos1_X),2)+EXPT((rReadfeedPos3_Y-rReadfeedPos1_Y),2)));;	
END_IF

IF (rReadfeedPos4_Y-rReadfeedPos1_Y)>=0 THEN
	rAngle_b:=360/(2*math.PI)*ACOS((rReadfeedPos4_X-rReadfeedPos1_X)/SQRT(EXPT((rReadfeedPos4_X-rReadfeedPos1_X),2)+EXPT((rReadfeedPos4_Y-rReadfeedPos1_Y),2)));
	rAngle_PI_b:=ACOS((rReadfeedPos4_X-rReadfeedPos1_X)/SQRT(EXPT((rReadfeedPos4_X-rReadfeedPos1_X),2)+EXPT((rReadfeedPos4_Y-rReadfeedPos1_Y),2)));
ELSE
	rAngle_b:=360-360/(2*math.PI)*ACOS((rReadfeedPos4_X-rReadfeedPos1_X)/SQRT(EXPT((rReadfeedPos4_X-rReadfeedPos1_X),2)+EXPT((rReadfeedPos4_Y-rReadfeedPos1_Y),2)));
	rAngle_PI_b:=2*math.PI-ACOS((rReadfeedPos4_X-rReadfeedPos1_X)/SQRT(EXPT((rReadfeedPos4_X-rReadfeedPos1_X),2)+EXPT((rReadfeedPos4_Y-rReadfeedPos1_Y),2)));;	
END_IF

rRotation_C:=(rAngle+rAngle_a+rAngle_b-135)/3;

C:=(rAngle_PI+rAngle_PI_a+rAngle_PI_b-135*math.PI/180)/3;
x0:=Tx:=rReadfeedPos1_X; y0:=Ty:=rReadfeedPos1_Y; Tz:=rReadfeedPos1_Z;
x1:=rReadfeedPos2_X; 	 y1:=rReadfeedPos2_Y;
x2:=rReadfeedPos3_X; 	 y2:=rReadfeedPos3_Y;
x3:=rReadfeedPos4_X; 	 y3:=rReadfeedPos4_Y;

Output_X0:=(y0-Ty)*SIN(C)+(x0-Tx)*COS(C);
Output_Y0:=(-x0+Tx)*SIN(C)+(y0-Ty)*COS(C);

Output_X1:=(y1-Ty)*SIN(C)+(x1-Tx)*COS(C);
Output_Y1:=(-x1+Tx)*SIN(C)+(y1-Ty)*COS(C);

Output_X2:=(y2-Ty)*SIN(C)+(x2-Tx)*COS(C);
Output_Y2:=(-x2+Tx)*SIN(C)+(y2-Ty)*COS(C);

Output_X3:=(y3-Ty)*SIN(C)+(x3-Tx)*COS(C);
Output_Y3:=(-x3+Tx)*SIN(C)+(y3-Ty)*COS(C);

dx:=((y1-y0+y2-y3)*SIN(C)/2+(-x0+x1+x2-x3)*COS(C)/2)/15;
dy:=((x0+x1-x2-x3)*SIN(C)/2+(-y0-y1+y2+y3)*COS(C)/2)/15;

END_FUNCTION_BLOCK

// Controller_3200C/Application/LogicControl
PROGRAM LogicControl
VAR_INPUT
	xReStart: BOOL;	
END_VAR
VAR
	CameraInterface			: L_RPP_CameraInterface;
	// CameraInterface
	ipAddr					: NBS.IP_ADDR:= ( sAddr := '192.168.5.20' );
	xAutoMode				: BOOL;
	xShootInternal			: BOOL;
	lrInternalTrigTime		: LREAL;
	xShootTrig				: BOOL;
	fb_TON_ReadStatus		: TON;
	xStatusInit				: BOOL;
	Read_TON      			: ARRAY [1..36] OF TON;
	ReadA1_Step				:INT;
	ReadA2_Step				:INT;
	ReadA3_Step				:INT;
	ReadAuxC_Step			:INT;
	iProd_Count				:INT;
END_VAR

	IF NOT xStatusInit THEN
		fb_TON_ReadStatus.IN:=TRUE;
		fb_TON_ReadStatus.PT:=T#5S;
	END_IF
	
	IF fb_TON_ReadStatus.Q THEN
		fb_TON_ReadStatus.IN:=FALSE;
		xStatusInit:=TRUE;
	END_IF
	 
	IF xStatusInit THEN
		A20_StatusDisplay();//设备状态
	END_IF

		
	A40_Modbus_Slave();	
	
(*******************************01——程序编辑*********************************) 
		A01_EditPrg();
(*******************************10——回零*********************************)
		A10_Homing();	
(*******************************40——参数设置*********************************)
		//A40_SetParameters();
(*******************************50——设置抱闸开关*********************************)	
		A50_Brake();
	
	
	IF iPrdtDetectDevice=Detect_Device.Camera THEN//产品检测装置选择 0：相机；1：传感器；2：上位机通讯指定
		xCameraEnable:=TRUE;
	ELSE
		xCameraEnable:=FALSE;
	END_IF
	IF iPrdtDetectDevice=Detect_Device.Sensor THEN//产品检测装置选择 0：相机；1：传感器；2：上位机通讯指定
		xSensorEnable:=TRUE;
	ELSE
		xSensorEnable:=FALSE;
	END_IF
	
	IF iPrdtDetectDevice=Detect_Device.Computer THEN//产品检测装置选择 0：相机；1：传感器；2：上位机通讯指定
		xComputerEnable:=TRUE;
	ELSE
		xComputerEnable:=FALSE;
	END_IF
	
	A10_CameraInterface();


	IF ModbusServer_1.byClientConnections<>0 AND NOT xInitWindow  THEN
		fb_TON2.IN:=TRUE;
		fb_TON2.PT:=T#200MS;
	END_IF
	
	IF fb_TON2.Q=TRUE THEN
		fb_TON2.IN:=FALSE;
		xInitWindow:=TRUE;		
		iHMI_InitWindow:=600;	

	END_IF	
		fb_TON2();
		fb_TON_ReadStatus();

ACTION A40_Modbus_Slave:
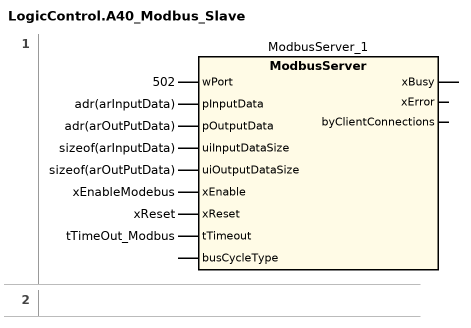
// NETWORK 1
ModbusServer_1(
    wPort := 502,
    pInputData := adr(arInputData),
    pOutputData := adr(arOutPutData),
    uiInputDataSize := sizeof(arInputData),
    uiOutputDataSize := sizeof(arOutPutData),
    xEnable := xEnableModebus,
    xReset := xReset,
    tTimeout := tTimeOut_Modbus); // ModbusServer

// NETWORK 2
END_ACTION

ACTION A20_StatusDisplay:
	

	
	//机器人各状态
	RobotAxesEnable:=	 	ReadAxisAuxCInfo.PowerOn AND ReadAxis1Info.PowerOn AND ReadAxis2Info.PowerOn AND ReadAxis3Info.PowerOn;	
	RobotAxesGroupEnable:=  Delta_Robot.xGroupEnable;
	RobotHoming:=			Delta_Robot.xAxesGroupIsHomed;	
	RobotSlimit	:=			Delta_Robot.pAxis_X^.xSWLimitNeg AND Delta_Robot.pAxis_X^.xSWLimitPos AND Delta_Robot.pAxis_Y^.xSWLimitNeg 
						AND Delta_Robot.pAxis_Y^.xSWLimitPos AND Delta_Robot.pAxis_Z^.xSWLimitNeg AND Delta_Robot.pAxis_Z^.xSWLimitPos;		
	RobotAxesWarning:=		Delta_Robot.xWarning;	//	Delta_Robot.xWarning
	RobotAxesError:=		Delta_Robot.xError;		//	Delta_Robot.xError
	RobotPrgOrParaError:= (ErrorID<>0);
	
	//旋转轴各状态		

	
	//A1轴各状态		
    A1axisEnable:=		        A1.xDriveEnabled;	 
    A1axisHoming:=		        ReadAxis1Info.IsHomed;
    A1axisSPlimit:=		        A1.xSWLimitPos;		
    A1axisSNlimit:=		        A1.xSWLimitNeg;		
    A1axis24Warning:=			NOT DO_3;    									
    A1axisWarning:=		        A1.xWarning;		
    A1axisError	:=		        A1.xError;	
	
	//A2轴各状态	
    A2axisEnable:=		    A2.xDriveEnabled;	                                        
    A2axisHoming:=		    ReadAxis2Info.IsHomed;                                                                           
    A2axisSPlimit:=		    A2.xSWLimitPos;		                                         
    A2axisSNlimit:=		    A2.xSWLimitNeg;		                                                                                  
    A2axis24Warning:=		NOT DO_3;									                                                   
    A2axisWarning:=		    A2.xWarning;		                                            
    A2axisError	:=		    A2.xError;	                                               
	
	//A3轴各状态
    A3axisEnable:=		    A3.xDriveEnabled;	                                        
    A3axisHoming:=		    ReadAxis3Info.IsHomed;                                                                             
    A3axisSPlimit:=		    A3.xSWLimitPos;		                                         
    A3axisSNlimit:=		    A3.xSWLimitNeg;		                                         		                                         
    A3axis24Warning:=		NOT DO_3;										                                                   
    A3axisWarning:=		    A3.xWarning;		                                            
    A3axisError	:=		    A3.xError;	                                               
	
	//外部错误输入信号
	IF NOT DI_4 THEN
	;//	ErrorID:=1111;
	END_IF

	
	//系统错误与警告	//modified in 2016.11.03
	xSystemError:=AGBControl.xAxesGroupError OR Delta_Robot.xError OR A1.xError OR A2.xError 
					OR A3.xError OR Axis_X.xError OR Axis_Y.xError OR Axis_Z.xerror OR ErrorID<>0 OR Aux1_ABC.xError ;//OR NOT DI_4;

	xSystemWarning:=AGBControl.xAxesGroupWarning OR Delta_Robot.xWarning OR A1.xWarning OR A2.xWarning OR Aux1_ABC.xDriveWarning 
					OR A3.xWarning  OR Axis_x.xWarning OR Axis_y.xWarning OR axis_z.xWarning OR WarningID<>0 OR CustomerPrgHandling.xWarning;
	//xSystemWarning:=CustomerPrgHandling.xWarning;
	
	//modified in 2016.11.03				
	xEmergencyStop:=A1.xDriveWarning OR A2.xDriveWarning OR A3.xDriveWarning ;
	
	//光电开关信号显示
	xPhoSwitch:=DI_3;
	//光电开关信号显示
	

	//modified in 2016.11.03
	IF AGBControl.xRegulatorOnALL  AND Aux1_ABC.xRegulatorOn THEN	//modified in 2016.11.03
		xLED1Status:=TRUE;
	END_IF
	
		//运行指示灯
	IF xSystemError THEN
		xLED1Status:=FALSE;
	END_IF
	
	
	//modified in 2016.11.03
	IF NOT AGBControl.xRegulatorOnALL AND NOT Aux1_ABC.xRegulatorOn AND NOT xSystemError  THEN
		
		IF NOT xLock_LED1 THEN
			LED1_TON1.IN:=TRUE;
			LED1_TON1.PT:=T#0.5S;
			IF LED1_TON1.Q THEN
				LED1_TON1.IN:=FALSE;
				xLED1Status:=TRUE;
				xLock_LED1:=TRUE;
			END_IF
		END_IF
		
		IF xLock_LED1 THEN
			LED1_TON2.IN:=TRUE;
			LED1_TON2.PT:=T#0.5S;
			IF LED1_TON2.Q THEN
				LED1_TON2.IN:=FALSE;
				xLED1Status:=FALSE;
				xLock_LED1:=FALSE;
			END_IF					
		END_IF
	END_IF
	
	LED1_TON1();
	LED1_TON2();

	//故障指示灯
	IF NOT xSystemError  AND NOT xSystemWarning THEN //无故障和警告时，常灭
		xLED2Status:=FALSE;
	END_IF
	
	IF xSystemError OR xSystemWarning THEN	//故障或警告时，常闪

		IF xSystemWarning THEN
			rLED2FlashTime:=250;
		END_IF
		
		IF xSystemError THEN
			rLED2FlashTime:=500;
		END_IF
		
		IF NOT xLock_LED2 THEN
			LED2_TON1.IN:=TRUE;
			LED2_TON1.PT:=REAL_TO_TIME(1000-rLED2FlashTime);
			IF LED2_TON1.Q THEN
				LED2_TON1.IN:=FALSE;
				xLED2Status:=TRUE;
				xLock_LED2:=TRUE;
			END_IF			
		END_IF
		
		IF xLock_LED2 THEN
			LED2_TON2.IN:=TRUE;
			LED2_TON2.PT:=REAL_TO_TIME(rLED2FlashTime);
			IF LED2_TON2.Q THEN
				LED2_TON2.IN:=FALSE;
				xLED2Status:=FALSE;
				xLock_LED2:=FALSE;
			END_IF					
		END_IF
		
	END_IF
	LED2_TON1();
	LED2_TON2();
	
	
	
	

